	Position	: REAL	:= 0.0;	(* Actual Position *)
	Velocity	: REAL	:= 0.0;	(* Actual Velocity *)
	Torque		: REAL	:= 0.0;	(* Actual Torque *)
	Error		: UDINT	:= 0;	(* Error Code *)
	PowerActive	: BOOL  := FALSE;
	
END_STRUCT
END_TYPE

// ---- Data types/TF/Palletizer/TFMachinePalletizer_GatesAccess.TcDUT
TYPE TFMachinePalletizer_GatesAccess :
STRUCT
	GateAccessConsolle 	: TFGateAccess; //Consolle
	GateAccessPS306 	: TFGateAccessNoStop; //PS306 - Lato Sx Inizio
	GateAccessPS307 	: TFGateAccessNoStop; //PS307 - Lato Sx Centrale
	GateAccessPS308		: TFGateAccessNoStop; //PS308 - Lato Dx Centrale
	GateAccessPS309		: TFGateAccessNoStop; //PS309 - Lato DX In Fondo
END_STRUCT
END_TYPE

// ---- Data types/TF/Palletizer/TFMachinePalletizer_ManCmd.TcDUT
TYPE TFMachinePalletizer_ManCmd :
STRUCT
	CyclePallet : BOOL;
	CycleLayer : BOOL;
	Dest : INT;
	
	CicloRiposo	: BOOL;
	StepCiclo	: bool;
END_STRUCT
END_TYPE

// ---- Data types/TF/Palletizer/TFMachinePalletizer_ParametersFromHMI.TcDUT
TYPE TFMachinePalletizer_ParametersFromHMI :
STRUCT

	OffsetKPick					: REAL;	(* Offset di apertura pinza per prelievo pallet, falda  *)
	OffsetKPickPack				: REAL;	(* Offset di apertura pinza per prelievo pacco *)
	OffsetKPlacePack			: REAL;	(* Offset di apertura pinza per deposito pacco *)
	OffsetKPlace				: REAL;	(* Offset di apertura pinza per deposito pallet *)
	OffsetZPlacePallet			: REAL;	(* Offset quota Z per rilascio pallet *)
	OffsetZPlaceLayer			: REAL;	(* Offset quota Z per rilascio falda *)
	
	KPickTorquePallet			: REAL;	(* Coppia per prelievo Pallet *)
	
	OffsetZPlacePaccoVerticale		: REAL	:= 0; (* Offset quota Z per rilascio pacco in verticale *)
	OffsetZPlacePaccoOrrizzontale	: REAL 	:= 0;	(* Offset quota Z per rilascio pacco in Orrizzontale *)
	
	OffsetZUscitaTasteggioPickPallet : REAL := 10; (* Offset dell'asse Z durante un tasteggio in prelievo Pallet: l'asse Z si muove di questo offset dopo la ri-lettura dei tastatori *)

END_STRUCT
END_TYPE

// ---- Data types/TF/Palletizer/TFMachinePalletizer_WorkAreaOffset.TcDUT
(* Offset di posizionamento, rispetto alla posizione assoluta, delle postazioni nelle varie direzioni*)
TYPE TFMachinePalletizer_WorkAreaOffset :
STRUCT
	X : REAL := 0;	//Offset in direzione X
	Y : REAL := 0;	//Offset in direzione Y
	Z : REAL := 0;	//Offset in direzione Z
	RX : REAL := 0;	//Offset di rotazione lungo X
	RY : REAL := 0;	//Offset di rotazione lungo Y
	RZ : REAL := 0;	//Offset di rotazione lungo Z
END_STRUCT
END_TYPE

// ---- Data types/TF/Palletizer/TFMachinePalletizer_WorkAreaSort.TcDUT
TYPE TFMachinePalletizer_WorkAreaSort :
STRUCT
	Distance : LREAL;
	cwa : UINT;
END_STRUCT
END_TYPE

// ---- Data types/TF/Palletizer/TFMachinePalletizer_WorkAreaZone.TcDUT
TYPE TFMachinePalletizer_WorkAreaZone :
STRUCT
	Zone		: ARRAY[1..MAXZONE] OF TFMachinePalletizer_Zone; (* Definizione Zone *)
END_STRUCT
END_TYPE

// ---- Data types/TF/Palletizer/TFMachinePalletizer_WorkPickPointState_OLD.TcDUT
TYPE TFMachinePalletizer_WorkPickPointState_OLD :
STRUCT
	
	State			: INT	:= 0;	(* Stato PickPoint (0=Pacco Assente, 1=Pacco Presente *)
	Code			: INT	:= 0;	(* Codice Pacco *)
	NextCode		: INT	:= 0;   (* Codice Pacco Successivo *)
	TC				: INT   := 0;   (* Comando Ribaltino 0=Nop, 1=Ribaltino Verticale, 2=Ribaltino Orizzontale *)
	TS				: INT	:= 0;   (* Stato Ribaltino; 0=Nop,1=Ribaltino Verticale, 2=Ribaltino Orizzontale *)
	NextTC			: INT	:= 0;   (* Comando Successivo Ribaltino; 0=Nop, 1=Ribaltino Verticale, 2=Ribaltino Orizzontale*)
	ZTilter			: REAL  := 0.0; (* Quota asse Ribaltino, Scritta dall'Handling *)
	Encumbrance		: BOOL	:= FALSE; (* TRUE:= Le dimensioni del pacco sono tali da impegnare anche la PX di Uscita del Deviatore, FALSE:= Pacco cCmpletamente sul Ribaltino*)
	
	XDim			: REAL;		(* (mm) Dimensione X del Pacco *)
	YDim			: REAL;		(* (mm) Dimensione Y del Pacco *)
	ZDim			: REAL;		(* (mm) Dimensione Z del Pacco *)
	
END_STRUCT
END_TYPE

// ---- Data types/TF/Palletizer/TFMachinePalletizer_WorkPPOffset.TcDUT
TYPE TFMachinePalletizer_WorkPPOffset :
STRUCT
	Xv	:	REAL := 0.0; (* READ	- (mm) Offset del punto di prelievo in direzione X per ribaltino verticale *)
	Yv	:	REAL := 0.0; (* READ	- (mm) Offset del punto di prelievo in direzione Y per ribaltino verticale *)
	Zv	:	REAL := 0.0; (* READ	- (mm) Offset del punto di prelievo in direzione Z per ribaltino verticale *)
	Jv	:	REAL := 0.0; (* READ	- (mm) Offset di rotazione J  per ribaltino verticale *)
	
	Xh	:	REAL := 0.0; (* READ	- (mm) Offset del punto di prelievo in direzione X per ribaltino orrizontale *)
	Yh	:	REAL := 0.0; (* READ	- (mm) Offset del punto di prelievo in direzione Y per ribaltino orrizontale *)
	Zh	:	REAL := 0.0; (* READ	- (mm) Offset del punto di prelievo in direzione Z per ribaltino orrizontale *)
	Jh	:	REAL := 0.0; (* READ	- (mm) Offset di rotazione J per ribaltino orrizontale  *)
END_STRUCT
END_TYPE

// ---- Data types/TF/Palletizer/TFMachinePalletizer_Zone.TcDUT
TYPE TFMachinePalletizer_Zone :
STRUCT
	
	WorkArea	: ARRAY[1..MAXAREA] OF INT; 			(* Numero delle WorkArea *)
	Code		: ARRAY[1..MAXFORMINGCODE] OF INT;		(* Codici di Pallettizzazione (0..n=, -1 dato non valido) *)
	
END_STRUCT
END_TYPE

// ---- Data types/TF/Palletizer/TFModulePalletizerRobot_TCPPar.TcDUT
TYPE TFModulePalletizerRobot_TCPPar :
STRUCT
	
	X	: LREAL := 0;	(* READ	- X Axe Parameters (UI Position=mm, UI Velocity=mm/sec UI Acc/Dec=mm/sec2) *)
	Y	: LREAL := 0;	(* READ	- Y Axe Parameters (UI Position=mm, UI Velocity=mm/sec UI Acc/Dec=mm/sec2) *)
	Z	: LREAL := 0;	(* READ	- Z Axe Parameters (UI Position=mm, UI Velocity=mm/sec UI Acc/Dec=mm/sec2) *)
	
END_STRUCT
END_TYPE

// ---- Data types/TF/Palletizer/TFModulePalletizerRobot_Point.TcDUT
TYPE TFModulePalletizerRobot_Point :
STRUCT
	
	X				: REAL	:= 0.0;	(* X Position *)
	Y				: REAL	:= 0.0;	(* Y Position *)
	Z				: REAL	:= 0.0;	(* Z Position *)
	J				: REAL	:= 0.0;	(* J Position *)
	
END_STRUCT
END_TYPE

// ---- Data types/TF/Palletizer/TFModulePalletizerRobot_ManCmd.TcDUT
TYPE TFModulePalletizerRobot_ManCmd :
STRUCT
	
	X	: TFMachinePalletizer_AxeManCmd;	(* X Axe Manual Command *)
	Y	: TFMachinePalletizer_AxeManCmd;	(* Y Axe Manual Command *)
	Z	: TFMachinePalletizer_AxeManCmd;	(* Z Axe Manual Command *)
	J	: TFMachinePalletizer_AxeManCmd;	(* J Axe Manual Command *)
	K	: TFMachinePalletizer_AxeManCmd;	(* K Axe Manual Command *)
	
	GeneralHome : BOOL;
	
	SuctionOn 	: BOOL;
	SuctionOff 	: BOOL;
	SuctionUp 	: BOOL;
	SuctionDown : BOOL;

	Pinza : TFMachinePalletizer_PinzaVentoseManCmd;
	
	PosizionamentoPinza0 	: BOOL; //Posizionamento pinza 0°
	PosizionamentoPinza90 	: BOOL; //Posizionamento pinza 90°
	PosizionamentoPinza180 	: BOOL; //Posizionamento pinza 180°

END_STRUCT
END_TYPE

// ---- Data types/TF/Palletizer/TFMachinePalletizer_AxeParameters.TcDUT
TYPE TFMachinePalletizer_AxeParameters :
STRUCT
	
	HomeDefine		: REAL	:= 0.0;	(* READ	- Home Define (Posizione di Azzeramento Encoder) *)
	HomePosition	: REAL	:= 0.0;	(* READ	- Home Position (Posizione di Home) *)
	MaxVelocity		: REAL	:= 0.0;	(* READ	- Max Velocity (Velocità Massima) *)
	MaxAcceleration	: REAL	:= 0.0;	(* READ	- Max Acceleration (Accelerazione Massima) *)
	MaxDeceleration	: REAL	:= 0.0;	(* READ	- Max Deceleration (Decelerazione Massima) *)
	MinPosition		: REAL	:= 0.0;
	MaxPosition		: REAL	:= 0.0;
	MaxTorque		: REAL	:= 0.0;
	ManSlowVelocity	: REAL	:= 0.0; (* READ - Manual Slow Velocity (% of MaxVelocity) *)
	ManFastVelocity	: REAL	:= 0.0; (* READ - Manual Fast Velocity (% of MaxVelocity) *)
	
END_STRUCT
END_TYPE

// ---- Data types/TF/Palletizer/TFMachinePalletizer_AxeManCmd.TcDUT
TYPE TFMachinePalletizer_AxeManCmd :
STRUCT
	
	Home	: BOOL	:= FALSE;	(* READ	- Home (Ricerca Posizione di Home) *)
	JogPos	: BOOL	:= FALSE;	(* READ	- Jog + *)
	JogNeg	: BOOL	:= FALSE;	(* READ	- Jog - *)
	JogFast	: BOOL	:= FALSE;	(* READ	- Jog +/- in Fast Speed *)
	
END_STRUCT
END_TYPE

// ---- Data types/TF/Palletizer/TFMachinePalletizer_AxeState.TcDUT
TYPE TFMachinePalletizer_AxeState :
STRUCT
	
	Position	: REAL	:= 0.0;	(* Actual Position *)
	Velocity	: REAL	:= 0.0;	(* Actual Velocity *)
	Torque		: REAL	:= 0.0;	(* Actual Torque *)
	Error		: UDINT	:= 0;	(* Error Code *)
	
END_STRUCT
END_TYPE

// ---- Data types/TF/Palletizer/TFModulePalletizerRobot_AxisPar.TcDUT
TYPE TFModulePalletizerRobot_AxisPar :
STRUCT
	
	X	: TFMachinePalletizer_AxeParameters;	(* READ	- X Axe Parameters (UI Position=mm, UI Velocity=mm/sec UI Acc/Dec=mm/sec2) *)
	Y	: TFMachinePalletizer_AxeParameters;	(* READ	- Y Axe Parameters (UI Position=mm, UI Velocity=mm/sec UI Acc/Dec=mm/sec2) *)
	Z	: TFMachinePalletizer_AxeParameters;	(* READ	- Z Axe Parameters (UI Position=mm, UI Velocity=mm/sec UI Acc/Dec=mm/sec2) *)
	J	: TFMachinePalletizer_AxeParameters;	(* READ	- J Axe Parameters (UI Position=°,  UI Velocity=°/sec  UI Acc/Dec=°/sec2) *)
	K	: TFMachinePalletizer_AxeParameters;	(* READ	- K Axe Parameters (UI Position=mm, UI Velocity=mm/sec UI Acc/Dec=mm/sec2) *)
	
END_STRUCT
END_TYPE

// ---- Data types/TF/Palletizer/TFMachinePalletizer_Forming_OLD.TcDUT
TYPE TFMachinePalletizer_Forming_OLD :
STRUCT
	
	Enable		: INT							:= -1;	(* READ			- Formatura Abilitata 0=no, 1=si, -1 dato non valido *)
	Code		: ARRAY[1..MAXFORMINGCODE] OF INT;		(* READ			- Codici di Pallettizzazione (0..n=, -1 dato non valido) *)
	Pallet		: INT							:= -1;	(* READ			- Tipo di pallet assegnato (0 = tipo 0, 1 = tipo 1, 2 = tipo 2,  …. , 0 / -1 dato non valido *)
	Layer		: INT							:= -1;	(* READ			- Tipo di falda dopo il pallet (0 = assente, 1 = tipo 1, 2 = tipo 2,  …. , -1 dato non valido *)
	NLayer		: INT							:= -1;	(* READ			- Numero di falde da depositare ad inizio pallettizzazione *)
	Tape		: INT							:= -1;	(* READ			- Da Nastrare (0=no, 1=si, -1= non valido) *)
	LGVAttr		: INT								:= -1;  (* READ			- Attributi LGV (0=no, 1=si, -1= non valido) *)
	
	PX			: REAL							:= 0.0;	(* READ			- (mm) Pack X Dimension - Dimensione X (valore nominale) del pacco ribaltato in posizione verticale(al momento definiti come orizzontali) *)
	PY			: REAL							:= 0.0;	(* READ			- (mm) Pack Y Dimension - Dimensione Y (valore nominale) del pacco ribaltato in posizione verticale *)
	PZ			: REAL							:= 0.0;	(* READ			- (mm) Pack Z Dimension - Dimensione Z (valore nominale) del pacco ribaltato in posizione verticale *)
	PIZ			: REAL							:= 0.0;	(* READ			- (mm) Pack Z Pick  Offset - Offset Prelievo in Z *)
	PLZ			: REAL							:= 0.0; (* READ			- (mm) Pack Z Place Offset - Offset Deposito in Z *)
	AX			: REAL							:= 0.0; (* READ			- (mm) Approach X Distance - Distanza Accostamento X *)
	AY			: REAL							:= 0.0; (* READ			- (mm) Approach Y Distance - Distanza Accostamento X *)
	AZ			: REAL							:= 0.0; (* READ			- (mm) Approach Z Distance - Distanza Accostamento X *)
	KLT			: REAL							:= 0.0;	(* READ			- (%)  Valore di Coppia in presa Longitudinale *)
	KTT			: REAL							:= 0.0;	(* READ			- (%)  Valore di Coppia in Presa Trasversale *)
	KM			: INT							:= 0;	(* READ			- Modo Presa Pacco: 1=Position, 2=Position+Torque *)

	PickPosition: INT							:= 0; 	(* READ 		- 0 = misto, 1 = verticale, 2 = orizzontale*)
	PackXP		: ARRAY[1..MAXFORMINGPACK] OF TFMachinePalletizer_FormingPack; (* Tabella Pacchi X Positiva - Usata quando la X di Prelievo è Maggiore rispetto la quota di destinazione "Posizione Pallet" *)
	PackXN		: ARRAY[1..MAXFORMINGPACK] OF TFMachinePalletizer_FormingPack; (* Tabella Pacchi X Negativa - Usata quando la X di Prelievo è Minore rispetto la quota di destinazione "Posizione Pallet" *)
	
	GUID		: UINT;
	RecipeCode 	: UINT;              (* codice Ricetta *)
	
END_STRUCT
END_TYPE

// ---- Data types/TF/Palletizer/TFMachinePalletizer_FormingPack_OLD.TcDUT
TYPE TFMachinePalletizer_FormingPack_OLD :
STRUCT
	
	JP			: INT							:= -1;	(* READ	- Tipo di presa (1 = Longitudinale (x), 0 = Trasversale (Y se Verticale, Z se Orizzontale), -1 = dato non valido) *)
	Grip		: INT							:= -1;	(* READ	- Tipo di presa (0 = Verticale, 1 = Orizzontale, -1 = dato non valido) *)
	Trajectory	: INT							:= -1;	(* READ	- Tipo di percorso (0, 1, 2, 3, …) (-1 dato non valido) *)
	Layer		: INT							:= -1;	(* READ	- Tipo di falda dopo il pacco (0 = assente, 1 = tipo 1, 2 = tipo 2,  …. , -1 dato non valido *)
	
	X			: REAL							:= 0.0;	(* READ	- (mm) Destination - Coordinata X *)
	Y			: REAL							:= 0.0;	(* READ	- (mm) Destination - Coordinata Y *)
	Z			: REAL							:= 0.0;	(* READ	- (mm) Destination - Coordinata Z *)
	J			: REAL							:= 0.0;	(* READ	- (°)  Destination - Coordinata J *)
	
END_STRUCT
END_TYPE

(*
//Trajectory :	
 1= standard deposito in diagonale
 2= standard deposito in diagonale specchiato rispetto x
 3=	standard deposito in diagonale specchiato rispetto y
 4= standard deposito in diagonale specchiato rispetto x e y


Layer : quando devo mettere la falda






*)

// ---- Data types/TF/Palletizer/TFMachinePalletizer_IN.TcDUT
TYPE TFMachinePalletizer_IN :
STRUCT
	Mode : Mode;
	
	PowerOk : BOOL;
	
	SensorAir : BOOL;
	Sensor24Volt : BOOL;
	
	PX_WorkArea : ARRAY [1..MAXAREA] OF BOOL;
	
	HandlingRun : BOOL;
	
	Y_BeltSafety : BOOL;
	Z_BeltSafety : BOOL;
	PX_GripPresence : BOOL;
			
	WD_Trasporti : BOOL; //Watch DOG da Trasporti
	
END_STRUCT
END_TYPE

// ---- Data types/TF/Palletizer/TFMachinePalletizer_Layer_OLD.TcDUT
TYPE TFMachinePalletizer_Layer_OLD :
STRUCT
	X			: REAL	:= 0.0;	(* READ	- (mm) Dimensione X *)
	Y			: REAL	:= 0.0;	(* READ	- (mm) Dimensione Y *)
	Z			: REAL	:= 0.0;	(* READ	- (mm) Dimensione Z *)
END_STRUCT
END_TYPE

// ---- Data types/TF/Palletizer/TFMachinePalletizer_OUT.TcDUT
TYPE TFMachinePalletizer_OUT :
STRUCT
	Run : BOOL;
	Warning : BOOL;
	Error : BOOL;
	Horn : BOOL;
	StartHorn : BOOL;

	PowerActive : BOOL;
	
	HomeDone : BOOL;
	
	StopTilterReq : BOOL;
	PowerOffTilterReq : BOOL;
	PowerOnTilterReq : BOOL;
	ResetTilterReq : BOOL;
	StartTilter : BOOL;
	
	ClockSegnalazioni : bool;//Clock per segnalazioni varie
	
	PowerActiveSIMULAZIONE : BOOL;
	
	ClockSegnalazioniAlternato	: BOOL;//Clock Segnalazioni  Alternato
	ResetSirenaSegnalazioni : BOOL; //Segnale di stop suoneria sirena 
END_STRUCT
END_TYPE

// ---- Data types/TF/Palletizer/TFMachinePalletizer_Pallet_OLD.TcDUT
TYPE TFMachinePalletizer_Pallet_OLD :
STRUCT
	X			: REAL	:= 0.0;	(* READ	- (mm) Dimensione X *)
	Y			: REAL	:= 0.0;	(* READ	- (mm) Dimensione Y *)
	Z			: REAL	:= 0.0;	(* READ	- (mm) Dimensione Z *)
END_STRUCT
END_TYPE

// ---- Data types/TF/Palletizer/TFMachinePalletizer_VelocityOverride.TcDUT
TYPE TFMachinePalletizer_VelocityOverride :
STRUCT
	
	Auto		: REAL	:= 0.0;	(* READ	- (%) In Auto *)
	Jog			: REAL	:= 0.0;	(* READ	- (%) In Jog *)
	Pack		: REAL	:= 0.0;	(* READ	- (%) With Pack   (Durante il deposito di un pacco  / con Pacco a bordo) *)
	Pallet		: REAL	:= 0.0;	(* READ	- (%) With Pallet (Durante il deposito di un Pallet / con Pallet a bordo) *)
	Layer		: REAL	:= 0.0;	(* READ	- (%) With Layer  (Durante il deposito di un Layer  / con Falda a bordo) *)
	PickRip		: REAL	:= 0.0; (* READ - (%) Grip Free (Durante il prelievo di un Layer, una Falda o un Pacco) *)
	
END_STRUCT
END_TYPE

// ---- Data types/TF/Palletizer/TFMachinePalletizer_WorkArea_OLD.TcDUT
TYPE TFMachinePalletizer_WorkArea_OLD :
STRUCT

	Enable			: INT	:= -1;	(* READ			- Postazione Abilitata 0=no, 1=si, -1 dato non valido *)
	Typology		: INT	:= -1;	(* READ			- Tipologia 1=Catasta Vuoti, 2=Pallet Singolo, 3=Falda, -1 dato non valido *)
	Pallet			: INT	:= -1;	(* READ			- Tipo di pallet assegnato (0 = tipo 0, 1 = tipo 1, 2 = tipo 2,  …. , 0 / -1 dato non valido. Usato se Typology=1 *)
	Layer			: INT	:= -1;	(* READ			- Tipo di falda dopo il pallet (0 = assente, 1 = tipo 1, 2 = tipo 2,  …. , -1 dato non valido. Usato se Typology=3 *)
	Code			: INT	:= -1;	(* READ/WRITE	- Codice di Pallettizzazione (0..n=, -1 dato non valido). Viene estratto dalla Forming se Jolly=1, altrimenti lo si riceve! *)
	Jolly			: INT	:= -1;	(* READ/WRITE	- (Definizione del Codice di Pall... A carico del PLC) (0=no, 1=si, -1= non valido) *)
	Learn_Z			: REAL	:= 0.0;	(* READ			- (mm) Quota inizio Apprendimento "TouchProbe" Cataste e Falde) (Quota assoluta di impianto DA ORIGINE *)
	Learned_Z		: REAL	:= 0.0; (* WRITE		- Quota rilevata durante apprendimento *)
	DoLearn_Z			: INT	:= -1;	(* READ/WRITE 	- Stato apprendimento 0=Disabilitato, 1=Abilitato da Eseguire, 2=Eseguito, -1 dato non valido *)
	Slow			: INT	:= -1;	(* READ			- Primo Pacco in Lento (0=no, 1=si, -1= non valido) *)
	Taped			: INT	:= -1;	(* READ/WRITE	- Nastratura eseguita. Determina espulsione! (0=non eseguita, 1=eseguita, -1= non valido) *)
	RefuseLGV       : BOOL	:= FALSE;	(* READ		- Abilitazione chiamata LGV a termine pallettizzazione - TRUE= Non chiama LGV quando pallet pieno, FALSE= viene eseguita richiesta LGV *)
	Initialize		: BOOL	:= FALSE; 	(* READ		- Deposito pallet e falda se prevista e non continua la pallettizzazione, TRUE= deposita pallet e falda e non continua pallettizzazione, FALSE= Esegue tutto il ciclo regolarmente*)
	
	X				: REAL	:= 0.0;	(* READ			- (mm) Quota assoluta di impianto DA ORIGINE *)
	Y				: REAL	:= 0.0;	(* READ			- (mm) Quota assoluta di impianto DA ORIGINE *)
	Z				: REAL	:= 0.0;	(* READ			- (mm) Quota assoluta di impianto DA ORIGINE *)
	J				: REAL	:= 0.0;	(* READ			- (°) Quota assoluta di impianto DA ORIGINE *)
	H				: REAL	:= 0.0; (* READ/WRITE	- (mm) Altezza Reale. Viene calcolata dal PLC dopo ogni prelievo (Vuoti o Falde) o deposito Pallet e durante la pallettizzazione *)
	HPL				: REAL	:= 0.0; (* READ/WRITE   - (mm) Altezza del pallett utilizzato + altezza layers utilizzati *)
	
	JPick			: REAL	:= 0.0;	(* READ			- (°) Quota rotazione pinza per prelievo (usata se la workarea è un magazziono pallet/falde) *)
	KPick			: REAL	:= 0.0;	(* READ			- (mm) Quota apertura pinza per prelievo (usata se la workarea è un magazziono pallet/falde) *)
	JPlace			: REAL	:= 0.0;	(* READ			- (°) Quota rotazione pinza per deposito pallet/falde *)
	
	LGV_Req			: INT	:= 0;	(* READ/WRITE	- Richiesta LGV (0=Nop, 1=Richiesta LGV, 2= Consenso Ingresso, -1= non valido) *)
	LGV_GetIn_GetOut: INT	:= -1;	(* WRITE		- Tipo Richiesta LGV  (0=Nop, 1=Richiesta Prelievo, 2= Richiesta Deposito, -1= non valido) *)	
	LGV_LetIn		: INT	:= -1;	(* READ			- Stato LGV (0=Nop, 1=Richiesta Ingresso, 2=Fine Ingresso, -1= non valido) *)
	LGV_Footprint	: INT	:= -1;	(* READ			- Presenza Ingombro Veicolo (0=Nessun Ingombro, 1=In Ingombro, -1= non valido) *)
	LGV_ReqAbort	: BOOL	:= FALSE; (* READ		- Aborto chimata LGV *)
	
	ProgressiveNr	: UDINT;
	
END_STRUCT
END_TYPE

// ---- Data types/TF/Palletizer/TFMachinePalletizer_WorkFootprint.TcDUT
TYPE TFMachinePalletizer_WorkFootprint :
STRUCT
	X			: REAL	:= 0.0;	(* READ	- (mm) Quota assoluta di impianto DA ORIGINE *)
	Y			: REAL	:= 0.0;	(* READ	- (mm) Quota assoluta di impianto DA ORIGINE *)
	Z			: REAL	:= 0.0;	(* READ	- (mm) Quota assoluta di impianto DA ORIGINE *)
	XDim		: REAL	:= 0.0;	(* READ	- (mm) Dimensione X *)
	YDim		: REAL	:= 0.0;	(* READ	- (mm) Dimensione Y *)
	ZDim		: REAL	:= 0.0;	(* READ	- (mm) Dimensione Z *)	
END_STRUCT
END_TYPE

// ---- Data types/TF/Palletizer/TFMachinePalletizer_WorkPickPoint_OLD.TcDUT
TYPE TFMachinePalletizer_WorkPickPoint_OLD :
STRUCT
	
	Xv					: REAL	:= 0.0;		(* READ	- (mm) Quota assoluta di impianto DA ORIGINE - CON RIBALTINO IN VERTICALE *)
	Yv					: REAL	:= 0.0;		(* READ	- (mm) Quota assoluta di impianto DA ORIGINE - CON RIBALTINO IN VERTICALE *)
	Zv					: REAL	:= 0.0;		(* READ	- (mm) Quota assoluta di impianto DA ORIGINE - CON RIBALTINO IN VERTICALE *)
	Jv					: REAL	:= 0.0;		(* READ	- (mm) Quota assoluta di impianto DA ORIGINE - CON RIBALTINO IN VERTICALE *)
	ZvRaise				: REAL  := 0.0; 	(* READ	- (mm) Quota di salita per uscire dall'ingombro - CON RIBALTINO IN VERTICALE *)
	
	Xh					: REAL	:= 0.0;		(* READ	- (mm) Quota assoluta di impianto DA ORIGINE - CON RIBALTINO IN ORIZZONTALE *)
	Yh					: REAL	:= 0.0;		(* READ	- (mm) Quota assoluta di impianto DA ORIGINE - CON RIBALTINO IN ORIZZONTALE *)
	Zh					: REAL	:= 0.0;		(* READ	- (mm) Quota assoluta di impianto DA ORIGINE - CON RIBALTINO IN ORIZZONTALE *)
	Jh					: REAL	:= 0.0;		(* READ	- (mm) Quota assoluta di impianto DA ORIGINE - CON RIBALTINO IN ORIZZONTALE *)
	ZhRaise				: REAL  := 0.0; 	(* READ	- (mm) Quota di salita per uscire dall'ingombro - CON RIBALTINO IN ORIZZONTALE *)
	
END_STRUCT
END_TYPE

// ---- Data types/TF/Palletizer/TFMachinePalletizer_WorkSpace.TcDUT
TYPE TFMachinePalletizer_WorkSpace :
STRUCT
	X			: REAL	:= 0.0;	(* READ	- (mm) Quota assoluta di impianto DA ORIGINE *)
	Y			: REAL	:= 0.0;	(* READ	- (mm) Quota assoluta di impianto DA ORIGINE *)
	Z			: REAL	:= 0.0;	(* READ	- (mm) Quota assoluta di impianto DA ORIGINE *)
END_STRUCT
END_TYPE

// ---- Data types/TF/Palletizer/TFModulePalletizerRobot_Status.TcDUT
TYPE TFModulePalletizerRobot_Status :
STRUCT
	
	X	: TFMachinePalletizer_AxeState;	(* X Axe State (UI Position=mm, UI Velocity=mm/sec UI Acc/Dec=mm/sec2) *)
	Y	: TFMachinePalletizer_AxeState;	(* Y Axe State (UI Position=mm, UI Velocity=mm/sec UI Acc/Dec=mm/sec2) *)
	Z	: TFMachinePalletizer_AxeState;	(* Z Axe State (UI Position=mm, UI Velocity=mm/sec UI Acc/Dec=mm/sec2) *)
	J	: TFMachinePalletizer_AxeState;	(* J Axe State (UI Position=°,  UI Velocity=°/sec  UI Acc/Dec=°/sec2) *)
	K	: TFMachinePalletizer_AxeState;	(* K Axe State (UI Position=mm, UI Velocity=mm/sec UI Acc/Dec=mm/sec2) *)
	
	GroupSegmentVelocity : LREAL;
	GroupSegmentID : UDINT;
	
	MachineAuto : BOOL;
	MachineRun : BOOL;
	MachineError : UDINT;
	MachineErrorExtra : UDINT;
	
	RobotError : UDINT;
	RobotErrorExtra : UDINT;

	
END_STRUCT
END_TYPE

// ---- Data types/TF/Palletizer/TFModulePalletizerRobot_IN.TcDUT
TYPE TFModulePalletizerRobot_IN :
STRUCT
	
	PX_Touch 			: BOOL;
	PX_TouchEmergency 	: BOOL;
	PX_SuctionCupsUp	: BOOL;
	PX_StackLayer		: BOOL;
	PX_StackPallet		: BOOL;
	PX_GripPresence		: BOOL;
	
	Y_BeltSafety		: BOOL;
	Z_BeltSafety		: BOOL;

END_STRUCT
END_TYPE

// ---- Data types/TF/Palletizer/TFModulePalletizerRobot_OUT.TcDUT
TYPE TFModulePalletizerRobot_OUT :
STRUCT

	EV_Suction			: BOOL;
	EV_SuctionCupsUp	: BOOL;
	EV_SuctionCupsDown	: BOOL;
	
END_STRUCT
END_TYPE

// ---- Data types/TF/Rulliere/Macchina/TFMachineTransportIN.TcDUT
TYPE TFMachineTransportIN :
STRUCT
	Mode : Mode;
	PowerOk : BOOL;
	SensorAir : BOOL;
	Sensor24Volt : BOOL;
END_STRUCT
END_TYPE

// ---- Data types/TF/Rulliere/Macchina/TFMachineTransportManCmd.TcDUT
TYPE TFMachineTransportManCmd :
STRUCT
END_STRUCT
END_TYPE

// ---- Data types/TF/Rulliere/Macchina/TFMachineTransportOUT.TcDUT
TYPE TFMachineTransportOUT :
STRUCT
	Run : BOOL;
	Warning : BOOL;
	Error : BOOL;
	Horn : BOOL;
	StartHorn : BOOL;

	PowerActive : BOOL;
	
	HomeDone : BOOL;
	
	ClockSegnalazioni : BOOL;//Clock per segnalazioni varie
	
END_STRUCT
END_TYPE

// ---- Data types/TF/Rulliere/Moduli/Cinghia/TFCinghiaManCmd.TcDUT
TYPE TFCinghiaManCmd :
STRUCT
	Ax 					: TFAxManCmd;
	ResetModulo 		: BOOL;
	Ax2 				: TFAxManCmd;
	AbilitaCmdTandem	: BOOL;
END_STRUCT
END_TYPE

// ---- Data types/TF/Rulliere/Moduli/Cinghia/TFCinghia_IN.TcDUT
TYPE TFCinghia_IN :
STRUCT
	
	FTC_Presenza1 			: BOOL; // Fotocellula Presenza 1 "INGRESSO"
	FTC_Presenza1Enable 	: BOOL; // Fotocellula Presenza 1 Abilitata
	
	FTC_Presenza2		 	: BOOL; // Fotocellula Presenza 2 "MEDIANA"
	FTC_Presenza2Enable 	: BOOL; // Fotocellula Presenza 2 Abilitata 
	
	FTC_Presenza3		 	: BOOL; // Fotocellula Presenza 3 "USCITA"
	FTC_Presenza3Enable		: BOOL; // Fotocellula Presenza 3 Abilitata 
	
	StopEsterno 		: BOOL;//Comando di stop rotazione dall'esterno
	ConsensoDaValle 	: BOOL;//Consenso rotazione per invio materiale a valle
	StopDaMacchina 		: BOOL;//Stop COmando da macchina, per tutti quei comandi che rimangono sempre in esecuzione
	
END_STRUCT
END_TYPE

// ---- Data types/TF/Rulliere/Moduli/Cinghia/TFBancoScelta_IN.TcDUT
TYPE TFBancoScelta_IN :
STRUCT
	
	FTC_Presenza1 			: BOOL; // Fotocellula Presenza 1 "INGRESSO"
	FTC_Presenza1Enable 	: BOOL; // Fotocellula Presenza 1 Abilitata
	
	FTC_Presenza2		 	: BOOL; // Fotocellula Presenza 2 "MEDIANA"
	FTC_Presenza2Enable 	: BOOL; // Fotocellula Presenza 2 Abilitata 
	
	FTC_Presenza3		 	: BOOL; // Fotocellula Presenza 3 "USCITA"
	FTC_Presenza3Enable		: BOOL; // Fotocellula Presenza 3 Abilitata 
	
END_STRUCT
END_TYPE

// ---- Data types/TF/Rulliere/Moduli/Cinghia/TFCinghia_OUT.TcDUT
TYPE TFCinghia_OUT :
STRUCT
		FTC_Presenza1 : BOOL;//Segnale della FTC 1 in senso marcia
		FTC_Presenza2 : BOOL;//Segnale della FTC 2 in senso marcia
		FTC_Presenza3 : BOOL;//Segnale della FTC 3 in senso marcia	
		
		ConsensoAMonte 			: BOOL;//Consenso scarico materiale per modulo a monte
		VelocitaUscitaAValle 	: REAL;//Velocità di rotazione per modulo a valle
		StopEsterno 			: BOOL;//comando di stop esterno per altri moduli
		RichiestaAValle			: bool;//Richiesta di scarico al modulo a valle

END_STRUCT
END_TYPE

// ---- Data types/TF/Rulliere/Moduli/Cinghia/TFCinghiaParameters.TcDUT
TYPE TFCinghiaParameters :
STRUCT
	ExtraLoadSpace 		: REAL := 100; //Spazio Extra per fermata su sensore in fase di carico	
	ExtraUnloadSpace 	: REAL := 200; //Spazio Extra per scarico rulliera 
	ExtraSpinta      	: real := 50; //Spazion aggiungiuntivo per spinta pallet in accoppiamento
	//Con Carico a bordo
	VelocitaCarico			: REAL := 20; // [%] Percentuale Velocità Con carico a bordo
	AccCarico				: REAL := 20; // [%] Percentuale Accelerazione Con carico a bordo
	DecCarico				: REAL := 20; // [%] Percentuale Decelerazione Con carico a bordo
	//Senza Carico a bordo
	VelocitaVuoto			: REAL := 50; // [%] Percentuale Velocità Senza carico a bordo 
	AccVuoto				: REAL := 50; // [%] Percentuale Accelerazione Senza carico a bordo
	DecVuoto				: REAL := 50; // [%] Percentuale Decelerazione Senza carico a bordo
	//Manulai
	VelocitaJog				: REAL := 50; // [%] Percentuale Velocità Manuale
	AccJog					: REAL := 50; // [%] Percentuale Accelerazione Manuale
	DecJog					: REAL := 50; // [%] Percentuale Decelerazione Manuale

	CorrezioneVelocitaInverter2PerTandem 		: REAL := 5;
	CorrezioneVelocitaInverter2PerTandemMonte 	: REAL := 5;

END_STRUCT
END_TYPE

// ---- Data types/TF/Rulliere/Moduli/Cinghia/TFBancoScelta_OUT.TcDUT
TYPE TFBancoScelta_OUT :
STRUCT
		FTC_Presenza1 : BOOL;
		FTC_Presenza2 : BOOL;
		FTC_Presenza3 : BOOL;	
		
		
END_STRUCT
END_TYPE

// ---- Data types/TF/Rulliere/Moduli/Cinghia/TFMoveParAXCinghia.TcDUT
TYPE TFMoveParAXCinghia :
STRUCT
	AccCarico				: REAL := 20; // [mm/s2] Accelerazione FASE carico 
	DecCarico				: REAL := 20; // [mm/s2] Decelerazione FASE carico 
	VelocitaCarico			: REAL := 20; // [mm/s] Velocità FASE carico 
	
	AccScarico				: REAL := 20; // [mm/s2] Accelerazione FASE scarico
	DecScarico				: REAL := 20; // [mm/s2] Decelerazione FASE scarico
	VelocitaScarico			: REAL := 20; // [mm/s] Velocità FASE scarico
	
	VelocitaVuoto			: REAL := 20; // [mm/s] Velocità Senza carico a bordo 
	AccVuoto				: REAL := 20; // [mm/s2] Accelerazione Senza carico a bordo
	DecVuoto				: REAL := 20; // [mm/s2] Decelerazione Senza carico a bordo

	JerkConCarico			: REAL := 99999; //Jerk Con carico
	JerkVuoto				: REAL := 99999; //Jerk a Vuoto

END_STRUCT
END_TYPE

// ---- Data types/TF/Rulliere/Moduli/RullieraPallet/TFAxCentratoreManCmd.TcDUT
TYPE TFAxCentratoreManCmd :
STRUCT
	
	Home	: BOOL	:= FALSE;	(* Home (Ricerca Posizione di Home) *)
	JogPos	: BOOL	:= FALSE;	(* Jog + *)
	JogNeg	: BOOL	:= FALSE;	(* Jog - *)
	JogFast	: BOOL	:= FALSE;	(* Jog +/- in Fast Speed *)
	
	EseguiApertura 		: BOOL := FALSE; (* Porta il centratore tutto aperto *)
	EseguiCentratura 	: BOOL := FALSE; (* Esegue il ciclo di centratura *)
	
END_STRUCT
END_TYPE

// ---- Data types/TF/Rulliere/Moduli/RullieraPallet/TFAxTraslazioneRulliera.TcDUT
TYPE TFAxTraslazioneRulliera :
STRUCT
	
	Home	: BOOL	:= FALSE;	(* Home (Ricerca Posizione di Home) *)
	JogPos	: BOOL	:= FALSE;	(* Jog + *)
	JogNeg	: BOOL	:= FALSE;	(* Jog - *)
	JogFast	: BOOL	:= FALSE;	(* Jog +/- in Fast Speed *)
	
	MoveToCarico : BOOL := FALSE; (* Vai a posizione di CARICO*)
	MoveToScarico : BOOL := FALSE; (* Vai a posizione di CARICO*)
	MoveToPrelievo1 : BOOL := FALSE; (* Vai a posizione di CARICO*)
	MoveToPrelievo2 : BOOL := FALSE; (* Vai a posizione di CARICO*)
	
END_STRUCT
END_TYPE

// ---- Data types/TF/Rulliere/Moduli/RullieraPallet/TFCentratoreManCmd.TcDUT
TYPE TFCentratoreManCmd :
STRUCT
	Ax : TFAxCentratoreManCmd;
	ResetModulo : bool;	
END_STRUCT
END_TYPE

// ---- Data types/TF/Rulliere/Moduli/RullieraPallet/TFCentratoreParameters.TcDUT
TYPE TFCentratoreParameters :
STRUCT
	SogliaCentraturaEseguita	: REAL := 20; //Spazio Extra per fermata su sensore in fase di centratura	
	AbilitaCentratore			: bool := true; //Abilitazione centratore
	
	//Chiusura
	VelocitaChiusura		: REAL := 20; // [%] Percentuale Velocità chiusura(fino a sensori)
	VelocitaPareggiatura	: REAL := 20; // [%] Percentuale Velocità pareggiatura
	AccChiusura				: REAL := 20; // [%] Percentuale Accelerazione chiusura
	DecChiusura				: REAL := 20; // [%] Percentuale Decelerazione chiusra
	//Apertura
	VelocitaApertura		: REAL := 100; // [%] Percentuale Velocità apertura 
	AccApertura				: REAL := 100; // [%] Percentuale Accelerazione apertura
	DecApertura				: REAL := 100; // [%] Percentuale Decelerazione apertura
	
	//Manulai
	VelocitaJog				: REAL := 50; // [%] Percentuale Velocità Manuale
	AccJog					: REAL := 50; // [%] Percentuale Accelerazione Manuale
	DecJog					: REAL := 50; // [%] Percentuale Decelerazione Manuale

END_STRUCT
END_TYPE

// ---- Data types/TF/Rulliere/Moduli/RullieraPallet/TFCentratoreStatus.TcDUT
TYPE TFCentratoreStatus :
STRUCT

	Homed 		: BOOL; //Home modulo eseguito
	Error 		: UDINT; //Errore mofulo
	ErrorExtra 	: UDINT; //Errore extra modulo
	PowerActive : BOOL; //Modulo in marcia
	
	Ax1_State : TFMachinePalletizer_AxeState_weintek; //Stato asse 1
	
	Px_Home : BOOL; //Sensore reset
	Px_Aperto : BOOL; //Sensore extracorsa aperto
	Px_Chiuso : BOOL; //Sensore extracorsa chiuso

	Px_TouchDX : BOOL; //Sensore bandella DX
	Px_TouchSX : BOOL; //Sensore Bandella SX
	
	CentratoreAperto : BOOL;//Indica che il centratore è aperto in fuori ingombro
	
END_STRUCT
END_TYPE

// ---- Data types/TF/Rulliere/Moduli/RullieraPallet/TFCentratore_IN.TcDUT
TYPE TFCentratore_IN :
STRUCT
	
	TouchDX	: BOOL; //Sensore Bandella DX 1
	TouchSX		: BOOL; //Sensore Bandella SX 1
	
	PX_Aperto : BOOL; //Sensore MASSIMA APERTURA 1
	PX_Chiuso : BOOL; //Sensosre MASSIMA CHIUSURA 1
	PX_Home   : BOOL; //Sensore HOME 1
		
END_STRUCT
END_TYPE

// ---- Data types/TF/Rulliere/Moduli/RullieraPallet/TFCentratore_OUT.TcDUT
TYPE TFCentratore_OUT :
STRUCT
	PosizioneAperta : BOOL; //Posizione centratore Aperta e fuori ingombro
	PosizioneChiusa : BOOL; //Posizione centratore Chiusa e in ingombro
	PosizioneIndefinita : BOOL; //Posizione centratore Indefinita	
	
	FuoriIngombroXCarico : BOOL;//Posizione che consente alla rulliera di caricare senza che l'elemento in transito collida col centratore
	FuoriIngombroXScarico : BOOL;//Posizione che consente alla rulliera di scaricare l'elemento senza problemi
		
	TuochDX_Filtrato : BOOL;//Segnale stato bandella DX 
	TuochSX_Filtrato : BOOL;//Segnale stato bandella SX  

	PosizioneUltimaCentratura : REAL := 1900;//Posizione ultima centratura
		
END_STRUCT
END_TYPE

// ---- Data types/TF/Rulliere/Moduli/RullieraPallet/TFMoveParAXCentratore.TcDUT
TYPE TFMoveParAXCentratore :
STRUCT
	AccChiusura				: REAL := 20; // [mm/s2] Accelerazione Chiusura
	DecChiusura				: REAL := 20; // [mm/s2] Decelerazione Chiusura
	VelocitaChiusura		: REAL := 20; // [mm/s] Velocità Chiusura
	VelocitaApertura		: REAL := 20; // [mm/s] Velocità Apertura
	AccApertura				: REAL := 20; // [mm/s2] Accelerazione Apertura
	DecApertura				: REAL := 20; // [mm/s2] Decelerazione Apertura
	Jerk					: REAL := 999999;
	MinChiusura				: REAL := 400; 	// Quota minima di posizionamento	
	MaxApertura				: REAL := 1000; // Quota massima di posizionamento

END_STRUCT
END_TYPE

// ---- Data types/TF/Rulliere/Moduli/RullieraPallet/TFMoveParAXRulliera.TcDUT
TYPE TFMoveParAXRulliera :
STRUCT
	AccCarico				: REAL := 20; // [mm/s2] Accelerazione CON carico 
	DecCarico				: REAL := 20; // [mm/s2] Decelerazione CON carico 
	VelocitaCarico			: REAL := 20; // [mm/s] Velocità CON carico 
	
	AccScarico				: REAL := 20; // [mm/s2] Accelerazione SENZA scarico
	DecScarico				: REAL := 20; // [mm/s2] Decelerazione SENZA scarico
	VelocitaScarico			: REAL := 20; // [mm/s] Velocità SENZA scarico
	
	VelocitaVuoto			: REAL := 20; // [mm/s] Velocità Senza carico a bordo 
	AccVuoto				: REAL := 20; // [mm/s2] Accelerazione Senza carico a bordo
	DecVuoto				: REAL := 20; // [mm/s2] Decelerazione Senza carico a bordo
	JerkCarico				: REAL := 99999; //Jerk Con carico
	JerkVuoto				: REAL := 99999; //Jerk a Vuoto

	VelocitaPareggiatura	: REAL := 20; // [mm/s] Velocità Senza carico a bordo 


END_STRUCT
END_TYPE

// ---- Data types/TF/Rulliere/Moduli/RullieraPallet/TFMoveParAXTraslazioneRulliera.TcDUT
TYPE TFMoveParAXTraslazioneRulliera :
STRUCT
	AccCarico				: REAL := 20; // [mm/s2] Accelerazione Con carico a bordo
	DecCarico				: REAL := 20; // [mm/s2] Decelerazione Con carico a bordo
	VelocitaCarico			: REAL := 20; // [mm/s] Velocità Con carico a bordo
	VelocitaVuoto			: REAL := 20; // [mm/s] Velocità Senza carico a bordo 
	AccVuoto				: REAL := 20; // [mm/s2] Accelerazione Senza carico a bordo
	DecVuoto				: REAL := 20; // [mm/s2] Decelerazione Senza carico a bordo
END_STRUCT
END_TYPE

// ---- Data types/TF/Rulliere/Moduli/RullieraPallet/TFRullieraManCmd.TcDUT
TYPE TFRullieraManCmd :
STRUCT
	Ax 					: TFAxManCmd;
	ResetModulo 		: BOOL;
	Ax2 				: TFAxManCmd;
	AbilitaCmdTandemRulliere	: BOOL;
END_STRUCT
END_TYPE

// ---- Data types/TF/Rulliere/Moduli/RullieraPallet/TFRullieraMobileManCmd.TcDUT
TYPE TFRullieraMobileManCmd :
STRUCT
	AxR : TFAxManCmd;
	AxR2 : TFAxManCmd;
	AxT	: TFAxTraslazioneRulliera;
	ResetModulo : BOOL;
END_STRUCT
END_TYPE

// ---- Data types/TF/Rulliere/Moduli/RullieraPallet/TFRullieraMobileStatus.TcDUT
TYPE TFRullieraMobileStatus :
STRUCT
	Homed 		: BOOL; //Home modulo eseguito
	Error 		: UDINT; //Errore modulo
	ErrorExtra 	: UDINT; //Errore extra modulo
	PowerActive : BOOL; //Modulo in marcia
		
	Ax1_State : TFMachinePalletizer_AxeState_weintek; //Stato asse 1
	Ax2_State : TFMachinePalletizer_AxeState_weintek; //Stato Asse 2

	AxT_State : TFMachinePalletizer_AxeState_weintek; //Stato Asse Traslazione
	
	Element : TFMachineTransportElementWeintek;
	ElementPresente : BOOL;
	Element2 : TFMachineTransportElementWeintek;
	Element2Presente : BOOL;
	
	FTC_1 : BOOL; //Sensore 1
	FTC_2 : BOOL; //Sensore 2			
	FTC_3 : BOOL; //Sensore 3

	Px_Positivo : BOOL;//Sensore Extra corsa Positivo
	Px_Negativo : BOOL;//Sensore Extra corsa Positivo

	PosizioneRulliera : UINT; //Indica la posizione della rulliera

	StatoComando : UDINT;//Inidca lo stato in cui si trova il modulo

END_STRUCT
END_TYPE

// ---- Data types/TF/Rulliere/Moduli/RullieraPallet/TFRullieraParameters.TcDUT
TYPE TFRullieraParameters :
STRUCT
	ExtraLoadSpace 		: REAL := 100; //Spazio Extra per fermata su sensore in fase di carico	
	ExtraUnloadSpace 	: REAL := 200; //Spazio Extra per scarico rulliera 
	ExtraSpinta      	: real := 50; //Spazion aggiungiuntivo per spinta pallet in accoppiamento
	//Con Carico a bordo
	VelocitaCarico			: REAL := 20; // [%] Percentuale Velocità Con carico a bordo
	AccCarico				: REAL := 20; // [%] Percentuale Accelerazione Con carico a bordo
	DecCarico				: REAL := 20; // [%] Percentuale Decelerazione Con carico a bordo
	//Senza Carico a bordo
	VelocitaVuoto			: REAL := 50; // [%] Percentuale Velocità Senza carico a bordo 
	AccVuoto				: REAL := 50; // [%] Percentuale Accelerazione Senza carico a bordo
	DecVuoto				: REAL := 50; // [%] Percentuale Decelerazione Senza carico a bordo
	//Manulai
	VelocitaJog				: REAL := 50; // [%] Percentuale Velocità Manuale
	AccJog					: REAL := 50; // [%] Percentuale Accelerazione Manuale
	DecJog					: REAL := 50; // [%] Percentuale Decelerazione Manuale

	CorrezioneVelocitaInverter2PerTandem 		: REAL := 5;
	CorrezioneVelocitaInverter2PerTandemMonte 	: REAL := 5;

END_STRUCT
END_TYPE

// ---- Data types/TF/Rulliere/Moduli/RullieraPallet/TFRullieraStatus.TcDUT
TYPE TFRullieraStatus :
STRUCT

	Homed 		: BOOL; //Home modulo eseguito
	Error 		: UDINT; //Errore modulo
	ErrorExtra 	: UDINT; //Errore extra modulo
	PowerActive : BOOL; //Modulo in marcia
		
	Ax1_State : TFMachinePalletizer_AxeState_weintek; //Stato asse 1
	Ax2_State : TFMachinePalletizer_AxeState_weintek; //Stato Asse 2
	
	Element : TFMachineTransportElementWeintek;
	ElementPresente : BOOL;
	Element2 : TFMachineTransportElementWeintek;
	Element2Presente : BOOL;
	
	FTC_1 : BOOL; //Sensore 1
	FTC_2 : BOOL; //Sensore 2			
	FTC_3 : BOOL; //Sensore 3

	StatoComando : UDINT;//Inidca lo stato in cui si trova il modulo
	
END_STRUCT
END_TYPE

// ---- Data types/TF/Rulliere/Moduli/RullieraPallet/TFRulliera_IN.TcDUT
TYPE TFRulliera_IN :
STRUCT
	
	FTC_Presenza1 			: BOOL; // Fotocellula Presenza 1 "INGRESSO"
	FTC_Presenza1Enable 	: BOOL; // Fotocellula Presenza 1 Abilitata
	
	FTC_Presenza2		 	: BOOL; // Fotocellula Presenza 2 "MEDIANA"
	FTC_Presenza2Enable 	: BOOL; // Fotocellula Presenza 2 Abilitata 
	
	FTC_Presenza3		 	: BOOL; // Fotocellula Presenza 3 "USCITA"
	FTC_Presenza3Enable		: BOOL; // Fotocellula Presenza 3 Abilitata 
	
END_STRUCT
END_TYPE

// ---- Data types/TF/Rulliere/Moduli/RullieraPallet/TFRulliera_OUT.TcDUT
TYPE TFRulliera_OUT :
STRUCT
		FTC_Presenza1 : BOOL;
		FTC_Presenza2 : BOOL;
		FTC_Presenza3 : BOOL;	
		
		
END_STRUCT
END_TYPE

// ---- Data types/TF/Rulliere/Moduli/RullieraPallet/TFTraslazioneRullieraParameters.TcDUT
TYPE TFTraslazioneRullieraParameters :
STRUCT
	QuotaRullieraCarico 	: REAL := 100; //Posizione Rulliera di ingresso materiale	
	QuotaRullieraScarico 	: REAL := 2000; //Posizione Rulliera di uscita materiale
	QuotaRullieraPrelievo1 	: REAL := 100; //Posizione Rulliera di prelievo 1
	QuotaRullieraPrelievo2 	: REAL := 2000; //Posizione Rulliera di prelievo 2
	//Con Carico a bordo
	VelocitaCarico			: REAL := 20; // [%] Percentuale Velocità Con carico a bordo
	AccCarico				: REAL := 20; // [%] Percentuale Accelerazione Con carico a bordo
	DecCarico				: REAL := 20; // [%] Percentuale Decelerazione Con carico a bordo
	//Senza Carico a bordo
	VelocitaVuoto			: REAL := 50; // [%] Percentuale Velocità Senza carico a bordo 
	AccVuoto				: REAL := 50; // [%] Percentuale Accelerazione Senza carico a bordo
	DecVuoto				: REAL := 50; // [%] Percentuale Decelerazione Senza carico a bordo

	//Manulai
	VelocitaJog				: REAL := 50; // [%] Percentuale Velocità Manuale
	AccJog					: REAL := 50; // [%] Percentuale Accelerazione Manuale
	DecJog					: REAL := 50; // [%] Percentuale Decelerazione Manuale

END_STRUCT
END_TYPE

// ---- Data types/TF/Rulliere/Moduli/RullieraPallet/TFTraslazioneRulliera_IN.TcDUT
TYPE TFTraslazioneRulliera_IN :
STRUCT
	PX_Positive : BOOL; //Sensore Positivo
	PX_Negative : BOOL; //Sensore Negativo
	PX_Home   : BOOL; //Sensore HOME 
END_STRUCT
END_TYPE

// ---- Data types/TF/Rulliere/Moduli/TFAxManCmd.TcDUT
TYPE TFAxManCmd :
STRUCT
	
	Home	: BOOL	:= FALSE;	(* Home (Ricerca Posizione di Home) *)
	JogPos	: BOOL	:= FALSE;	(* Jog + *)
	JogNeg	: BOOL	:= FALSE;	(* Jog - *)
	JogFast	: BOOL	:= FALSE;	(* Jog +/- in Fast Speed *)
	
END_STRUCT
END_TYPE

// ---- Data types/TF/Rulliere/Moduli/TFAxParameters.TcDUT
TYPE TFAxParameters :
STRUCT
	HomeDefine		: REAL	:= 0.0;	(* Home Define (Posizione di Azzeramento Encoder) *)
	HomePosition	: REAL	:= 0.0;	(* Home Position (Posizione di Home) *)
	Vel				: REAL	:= 0.0;	(* Velocità di funzionamento*)
	Acc				: REAL	:= 100.0; (* Accelerazione di funzionamento *)
	Dec				: REAL	:= 100.0; (* Decelerazione di funzionamento *)
	Jerk			: REAL  := 100.0; (* Jerk di funzionamento *) 
	MaxTorque		: REAL	:= 100.0; (* Coppia massima utilizzata se si effettua il controllo di coppia*)
	JOGVel			: REAL	:= 100.0; (* Velocità JOG *)
	JOGAcc			: REAL	:= 100.0; (* Accelerazione JOG *)
	JOGDec 			: REAL	:= 100.0; (* Decelerazione JOG *)
	MaxDeceleration : REAL  := 100.0; (* Massima Decelerazione *)
	MinPosition		: REAL	:= 0.0;
	MaxPosition		: REAL	:= 0.0;
	MaxVel		    : REAL  := 0.0; (* Massima velocità per gestire i jog manuali *)
	MaxAcc		    : REAL  := 0.0; (* Massima velocità per gestire i jog manuali *)
	MaxDec		    : REAL  := 0.0; (* Massima velocità per gestire i jog manuali *)
	ManSlowVel		: REAL	:= 0.0; (* Manual Slow Velocity (% of MaxVelocity) *)
	ManFastVel		: REAL	:= 0.0; (* Manual Fast Velocity (% of MaxVelocity) *)
	Quota_Destinazione	: LREAL  := 0.0; (*Posizione target da raggiungere*)
	HomeVelocity		: REAL  := 1.0; (* Velocità per ricerca sesore di Home *)
END_STRUCT
END_TYPE

// ---- Data types/TF/Rulliere/Moduli/TFPortaStatus.TcDUT
TYPE TFPortaStatus :
STRUCT
	PortaAperta 	: BOOL;
	PortaChiusa 	: BOOL;
	AnomaliaPorta 	: BOOL;
END_STRUCT
END_TYPE

// ---- Data types/TF/Rulliere/Moduli/TFPortaManCmd.TcDUT
TYPE TFPortaManCmd :
STRUCT
	ApriPorta : BOOL;
	ChiudiPorta : bool;
END_STRUCT
END_TYPE

// ---- Data types/TF/Rulliere/Moduli/TFGestioneFTC_Misura_OUT.TcDUT
TYPE TFGestioneFTC_Misura_OUT :
STRUCT
	FTC_ZoccoloBassoFiltrata 	: BOOL;
	FTC_PallettoneFiltrata   	: BOOL;
	FTC_CavallinaBassaFiltrata 	: BOOL;
	FTC_CavallinaAltaFiltrata 	: BOOL;		

	LunghezzaMisurata 	: REAL;

	Supporto : TFMachinePalletizer_Pallet;
	
	MisuraInCorso : BOOL;
	MisuraDone : BOOL;
	
END_STRUCT
END_TYPE

// ---- Data types/TF/Rulliere/Moduli/TFBarcodeStatus.TcDUT
TYPE TFBarcodeStatus :
STRUCT

	Error 		: UDINT; //Errore modulo
	ErrorExtra 	: UDINT; //Errore extra modulo
		
	StatoLettore : StatusDataLogic;//Stato del lettore barcode

END_STRUCT
END_TYPE

// ---- Data types/TF/Rulliere/Moduli/TFTransportModules.TcDUT
TYPE TFTransportModules :
STRUCT

	BancoScelta 			: TFModuleSorterBancoScelta2Motori;
	ModuloCinghie 			: ARRAY[1..6] OF TFModuleCinghia;
	Bancalino 				: ARRAY[1..2] OF TFModuleBancalino;
	RullieraDopoBancalino 	: ARRAY[1..2] OF TFModuleRulliera;
	RullieraPareggiatore 	: ARRAY[1..2] OF TFModuleRulliera;
	RullieraPrelievo 		: ARRAY[1..2] OF TFModuleRulliera;
	
END_STRUCT
END_TYPE

// ---- Data types/TF/Rulliere/Moduli/TFTransportModuleStatus.TcDUT
TYPE TFTransportModuleStatus :
STRUCT
	Homed : BOOL; //Home modulo eseguito
	Error : UDINT;
	ErrorExtra : UDINT;
	PowerActive : BOOL; //Modulo in marcia
END_STRUCT
END_TYPE

// ---- Data types/TF/Rulliere/TFDimensionElement.TcDUT
TYPE TFDimensionElement :
STRUCT
	(* Dimensioni *)
	XDim		: REAL							:= 0.0;	(* (mm) Dimensione X *)
	YDim		: REAL							:= 0.0;	(* (mm) Dimensione Y *)
	ZDim		: REAL							:= 0.0;	(* (mm) Dimensione Z *)
END_STRUCT
END_TYPE

// ---- Data types/TF/Rulliere/TFMachinePalletizer_Pallet_Weintek.TcDUT
TYPE TFMachinePalletizer_Pallet_Weintek :
STRUCT
	Tipologia	: INT	:= -1;  (* Indica la tipologia dell'elemento *)
	Code		: INT;	(* Codici Della *)
	XDim		: REAL	:= 0.0;	(* (mm) Dimensione X *)
	YDim		: REAL	:= 0.0;	(* (mm) Dimensione Y *)
	ZDim		: REAL	:= 0.0;	(* (mm) Dimensione Z Base Cavallina o Base Cassa *)
	HMAX		: REAL  := 0.0;	(* (mm) Altezza Massima dell'elemento telaio cavallina o sponde cassa *)
	
	AltezzaDenteRitenuta	: REAL := 0.0; 	(* (mm) Altezza del dente di ritenuta (per cavalletti) *)
	Spessore_DenteRitenuta	: REAL := 0.0;	(* (mm) Spessore del dente di ritenuta (per cavalletti) *)
	OffsetY_DenteRitenuta 	: REAL := 0.0;	(* (mm) Posizione del dente di ritenuta rispetto la quota Y del cavalletto (per cavalletti) *)
	
	OFSDE_X90 				: REAL := 0.0;	(* (mm) OFFSET di deposito direzione X, utilizzato per PALLET o CASSE *)
	OFSDE_Y90 				: REAL := 0.0;	(* (mm) OFFSET di deposito direzione Y, utilizzato per PALLET o CASSE *)
	OFSDE_Z90 				: REAL := 0.0;	(* (mm) OFFSET di deposito direzione Z, utilizzato per PALLET o CASSE *)
	OFSDE_J90 				: REAL := 0.0;	(* (mm) OFFSET di deposito direzione J, utilizzato per PALLET o CASSE *)
	
	OFSDE_X0 				: REAL := 0.0;	(* (mm) OFFSET di deposito direzione X, utilizzato per CAVALLETTI *)
	OFSDE_Y0 				: REAL := 0.0;	(* (mm) OFFSET di deposito direzione Y, utilizzato per CAVALLETTI *)
	OFSDE_Z0 				: REAL := 0.0;	(* (mm) OFFSET di deposito direzione Z, utilizzato per CAVALLETTI *)
	OFSDE_J0 				: REAL := 0.0;	(* (mm) OFFSET di deposito direzione J, utilizzato per CAVALLETTI *)
	
	OFSDE_X180 				: REAL := 0.0;	(* (mm) OFFSET di deposito direzione X, utilizzato per CAVALLETTI *)
	OFSDE_Y180 				: REAL := 0.0;	(* (mm) OFFSET di deposito direzione Y, utilizzato per CAVALLETTI *)
	OFSDE_Z180 				: REAL := 0.0;	(* (mm) OFFSET di deposito direzione Z, utilizzato per CAVALLETTI *)
	OFSDE_J180 				: REAL := 0.0;	(* (mm) OFFSET di deposito direzione J, utilizzato per CAVALLETTI *)

	ConfigurazioneBC 	 : INT := -1;	(* (mm) Indica la modalità di funzionamento del barcode.. sono i suoi parametri *)
	QuotaRilevamentoBC_X : REAL := 0;	(* (mm) Indica la posizione del barcode lungo la sua lunghezza e rispetto il punto medio *)
	QuotaRilevamentoBC_Y : REAL := 0;	(* (mm) Indica la posizione del barcode lungo la sua larghezza e rispetto il punto medio	*)
	QuotaRilevamentoBC_Z : REAL := 0;	(* (mm) Indica la posizione del barcode lungo il suo spessore e rispetto il punto medio *)
	QuotaRilevamentoBC_J : REAL := 0;	(* (mm) Indica la posizione del barcode lungo il suo spessore e rispetto il punto medio *)

END_STRUCT
END_TYPE

// ---- Data types/TF/Rulliere/TFMachineTransportElement.TcDUT
TYPE TFMachineTransportElement :
STRUCT
	
	IDElement 		: UDINT := 0; //ID univoco generato dalla macchina  per il tracking degli alementi
	Barcode			: STRING := ''; //Barcode elemento
	DataElementOk 	: BOOL := FALSE;///Indica che i dati sono stati acquisiti e sono ok
	DataElement 	: TFMachinePalletizer_DataElement;
	DimElement 		: TFDimensionElement; //Dimensioni 
	Supporto		: TFMachinePalletizer_Pallet; (* Struttura del supporto presente sul punto di prelievo *)
	Zone			: e_ElementZone := e_ElementZone.NULL; //Zona di appartenenza dell'elemento
	ErrorAck		: BOOL := FALSE;//Se true, si attende un comando da parte dell'opperatore per far ripartire il ciclo
	CentraturaEsterna : e_StatoCentratura := CENTRATURA_DA_ESEGUIRE; //Stato della centratura estarna
	CentraturaInterna : e_StatoCentratura := CENTRATURA_DA_ESEGUIRE; //Stato della centratura interna
	Empty 				: BOOL := FALSE;	//Se TRUE significa che l'elemento è un vuoto
END_STRUCT
END_TYPE

// ---- Data types/TF/Rulliere/TFMachineTransportElementWeintek.TcDUT
TYPE TFMachineTransportElementWeintek :
STRUCT
	
	IDElement 		: UDINT := 0; //ID univoco generato dalla macchina  per il tracking degli alementi
	Barcode			: STRING := '';
	DataElementOk 	: BOOL := FALSE;///Indica che i dati sono stati acquisiti e sono ok
	DataElement 	: TFMachinePalletizer_DataElement;
	DimElement 		: TFDimensionElement; //Dimensioni 
	Supporto		: TFMachinePalletizer_Pallet_Weintek; (* Struttura del supporto presente sul punto di prelievo *)
	Zone			: INT := 0; //Zona di appartenenza dell'elemento
	ErrorAck		: BOOL := FALSE;//Se true, si attende un comando da parte dell'opperatore per far ripartire il ciclo
	CentraturaEsterna : INT; //Stato della centratura estarna
	CentraturaInterna : INT; //Stato della centratura interna
	Empty 			  : BOOL := FALSE;	//Se TRUE significa che l'elemento è un vuoto
END_STRUCT
END_TYPE

// ---- Data types/TF/Rulliere/TFMachineTransport_GatesAccess.TcDUT
TYPE TFMachineTransport_GatesAccess :
STRUCT
		
	GateAccessCarico 			: TFGateAccess;
	GateAccessCentratoreEsterno	: TFGateAccess;
	
END_STRUCT
END_TYPE

// ---- POUs/TFModules/DataBase/Record_From_DB.TcDUT
TYPE Record_From_DB :
STRUCT
	Udc 			: STRING(20);
	ArticleCode 	: STRING(20);
	Choice 			: STRING(5);
	Tone 				: STRING(5);
	Caliber 			: STRING(5);
	Length_mm 			: DINT;
	Width_mm 			: DINT;
	Thickness_mm 		: DINT;
	Quantity  			: LREAL;
	ArticleDescription 	: STRING(50);
END_STRUCT
END_TYPE

// ---- POUs/TFModules/DataBase/StoredProcedureState.TcDUT
TYPE StoredProcedureState :
STRUCT
	NumeroRecordLetti	: UDINT;//Numero di record letti
	ReadRun 		: BOOL;//Lettura in corso
	ReadDone 		: BOOL;//Lettura terminata con successo
	Error 			: BOOL;//Errore lettura
	ErrorID 		: UDINT;//ID Errore
	Sqlstate		: ST_DBSQLError;//State SQL
END_STRUCT
END_TYPE

// ---- POUs/TFModules/Misurazione Ingresso/TFGestioneFTC_Misura_IN.TcDUT
TYPE TFGestioneFTC_Misura_IN :
STRUCT
	FTC_ZoccoloBasso 	: BOOL;
	FTC_Pallettone   	: BOOL;
	FTC_CavallinaBassa 	: BOOL;
	FTC_CavallinaAlta 	: BOOL;
END_STRUCT
END_TYPE

// ---- Global Variables/BarCode/BarCODE.TcGVL
{attribute 'Tc2GvlVarNames'}
VAR_GLOBAL CONSTANT
	MAXNUMBARCODE		: INT := 4;		(* Identifica il numero dei BARCODE presenti nella WA (uno per ogni cassa nella WA) valorizza l'array dei BARCODE nella WASTATE *)
	DIMBARCODE			: INT := 13; 	(* Identifica la lunghezza del BARCODE *)

	(* Stati BARCODE *)
	LETTURA_DA_ESUGUIRE : INT := 0; 
	LETTURA_IN_CORSO 	: INT := 1;
	LETTURA_ESEGUITA 	: INT := 2;
	ERRORE				: INT := 3;
	
END_VAR

// ---- Global Variables/Comandi_1.TcGVL
{attribute 'Tc2GvlVarNames'}
VAR_GLOBAL CONSTANT
	
	CmdSbloccaBascolante 					: INT := 5000; (* Command: Do *)
	CmdBloccaBascolante 					: INT := 5100; (* Command: Do *)
	CmdSbloccaRotazione 					: INT := 5200; (* Command: Do *)
	CmdBloccaRotazione 						: INT := 5300; (* Command: Do *)
	CmdBloccaPinza							: INT := 5400; //blocco di tutta la pinza
	CmdSbloccaPinza							: INT := 5500; //sblocco di tutta la pinza

	
	StateSbloccaBascolante_RUN 			: INT := 5000;
	StateSbloccaBascolante_END 			: INT := 5099;
	StateBloccaBascolante_RUN 			: INT := 5100;
	StateBloccaBascolante_END 			: INT := 5199;
//                                        
	StateSbloccaRotazione_RUN 			: INT := 5200;
	StateSbloccaRotazione_END 			: INT := 5299;
	StateBloccaRotazione_RUN 			: INT := 5300;
	StateBloccaRotazione_END 			: INT := 5399;
                                          
	StateBloccaPinza_RUN 			: INT := 5400;
	StateBloccaPinza_END 			: INT := 5499;
	StateSbloccaPinza_RUN 			: INT := 5500;
	StateSbloccaPinza_END 			: INT := 5599;

	
END_VAR

// ---- Global Variables/Configurazione Impianto/Configurazione_Impianto.TcGVL
{attribute 'Tc2GvlVarNames'}
VAR_GLOBAL PERSISTENT
	(***********************************************************************************************************************************************************************************)
	(* Configurazioni comuni *)
	(***********************************************************************************************************************************************************************************)
	VERSO_PALLETTIZZATORE 				: e_Verso_Pallettizzatore 	:= PALLETTIZZATORE_SX; //Verso Pallettizzatore: stabilito guardando il pallettizzatore con la linea alle spalle
	TIPO_MAGAZZINO_FALDE  				: e_Tipo_Magazzino_Falde 	:= MAGAZZINO_FALDE_IN_WA; //Identifica il tipo di magazzino falde: MAGAZZINO_FALDE_CENTRO_FISSO = LA Y DI PRELIEVO RIMANE COSTANTE PER OGNI FORMATO,MAGAZZINO_FALDE_CENTRO_VARIABILE=LA Y DI PRELIEVO SI ADATTA AL FORMATO DELLA FALDA
	(***********************************************************************************************************************************************************************************)
	(* SOLO PER PALLETTIZZATORE LASTRE *)
	(***********************************************************************************************************************************************************************************)
	RIFERIMENTO_POSTAZIONE_WA			: e_RiferimentoPostazione 	:= CENTRALE; (*
												= 0		Identifica che la fotocellula di presenza della WorkArea è disposta sulla mediana della WorkArea stessa 	
												= 1 	Identifica che la fotocellula di presenza della WorkArea è disposta nell'angolo a SX della WorkArea stessa *)
	TIPOLOGIA_FUNZIONAMENTO_MACCHINA	: e_Tipo_Funzionamento := FUNZIONAMENTO_PICKING; (* Identifica la Tipolgia di funzionamento della Macchina *)											
	(***********************************************************************************************************************************************************************************)
	(* SOLO PER PALLETTIZZATORE PACCHI *)
	(***********************************************************************************************************************************************************************************)
	CATASTA_VUOTI_CON_RISCONTRI_FISSI 	: BOOL 						:= FALSE;	(*Se TRUE Identifica la presenza di riscontri fissi nella catasta dei vuoti (riscontri di centraggio) *)
	TIPO_RIBALTINO		  				: e_Tipo_Ribaltino 			:= RIBALTINO_DIRETTO;   (* Identifica il tipo di ribaltino (1= RIBALTINO DOPO SQUADRO,2= RIBALTINO DIRETTO) *)
	NPOSTAZIONE_DOPODELPUNTODIPREL		: UINT 						:= 5;		(* Numero Postazione DOPO del ribaltino ordine crescente di numero *)
	NPOSTAZIONE_PRIMADELPUNTODIPREL		: UINT 						:= 4;		(* Numero Postazione PRIMA del ribaltino, orfdine decrescente *)
	NumPostazionePALLET 				: INT; 									(* Indica il numero di postazione dove sono presenti I PALLET VUOTI *)
	(***********************************************************************************************************************************************************************************)
	(***********************************************************************************************************************************************************************************)
	NumPostazioneFALDE 					: UINT := 2; 							(* Indica il numero di postazione dove sono presenti LE FALDE *)
	NumPostazioneDiPareggiatura			: UINT := 3;							(* Indica il numero di postazione dove è presente la tavola di Pareggiatura *)

	ASSE_DISPOSIZIONE_POSTAZIONI		: e_Disposizione_Postazioni := LUNGO_X; (* Indica la disposizione delle postazioni rispeto gli assi della macchina, serve per capire la ciclica della macchina senza andare in collisione con le postazioni *)

	NUMERO_MACCHINA : UINT := 1; //Indica il numero della macchina in un impianto che usa la stessa HMI per discriminare eventuali pagine o funzioni in comune 

	ORDINE_DISPOSIZIONE_POSTAZIONI : e_OrdinamentoPostazione;// Indica come sono ordinate le postazioni rispetto l'origine della macchina: CRESCENTE o DECRESCENTE

	MAXAREAPRESENT : UINT := 4;//Piazzole di lavoro EFFETTIVAMENTE PRESENTI

	AngoloInclinazioneTavolaPareggiatura : REAL := 7; //Angolo in ° di inclinazione del della tavola di pareggiatura

	NumPostazioneBundle 	: UINT := 8;//Numero della postazione dedicata al bundle	
	AngoloInclinazioneBundle : REAL := 7; //Angolo in ° di inclinazione del del bundle

	NumPostazioneDeposito 	: UINT := 2;//Numero della postazione dedicata al deposito del materiale per pal picking
	NumPostazioneSuRulliera	: UINT := 1;//Numero della postazione dedicata al deposito del materiale per pal picking posizionata sulla rulliera
	

	
	HMaxScarto 			: REAL := 250;//Altezza massima ammissibile sul pancone degli scarti 
	CodeWasteSupport 	: INT := 4;	//Codice "Pallet dedicato al supporto degli scarti"
	
	TIPOLOGIA_RULLIERA_PRELIEVO : e_Tipologia_Rul_Prel;//Tipologia della ruliera di prelievo
	HMinFalde 			: REAL := 30;//Altezza minima sotto alla quale si manda in espulsione il pancone delle falde 
	CodeLayerSupport 	: INT := 15;	//Codice "Pallet dedicato al supporto delle falde"
	CodeWasteSlab		: INT := 3;//Codice lastra da scarare

	OFFSET_POSTAZIONE_LEGNO  : REAL := 680;//Offset filo fisso per legni rispetto al filo del bundle che è la quota di riferimento della WORKAREA lungo Y
	OFFSET_POSTAZIONE_TELAIO : REAL := 2630;//Offset filo fisso per TELAI rispetto al filo del bundle che è la quota di riferimento della WORKAREA lungo Y
	
	INGOMBRO_RISCONTRO_BUNDLE : REAL := 200;//Dimensione riscontro FISSO BUNDLE 
	INGOMBRO_RISCONTRO_FRAME : REAL := 100;//Dimensione riscontro FISSO BUNDLE 
END_VAR

VAR_GLOBAL CONSTANT

	(***********************************************************************************************************************************************************************************)
	(* SOLO PER PALLETTIZZATORE LASTRE *)
	(***********************************************************************************************************************************************************************************)
	//MAXPICKPOINTSTORE					: INT := 1;	(* Numero massimo di Punti di Prelievo di tipo Magazzino Falda *)
	//MAXPICKPOINTROLLER					: INT := 2;	(* Numero massimo di Punti di Prelievo di Tipo Rulliera *)
	(***********************************************************************************************************************************************************************************)
	(* SOLO PER PALLETTIZZATORE PACCHI *)
	(***********************************************************************************************************************************************************************************)
	ALTEZZA_CATASTA_VUOTI				: REAL := 1250;	(* Altezza Catasta Vuoti *)
	ALTEZZA_CATASTA_FALDE				: REAL := 900;	(* Altezza Catasta Falde *)
	
	DISTANZA_FTC_PINZA	: REAL := 650; (* Distanza tra le due fotocellule KEINCE sulla pinza *)

END_VAR

// ---- Global Variables/Errori/Errori_BarCODE.TcGVL
{attribute 'Tc2GvlVarNames'}
VAR_GLOBAL CONSTANT
	(* Errori BARCODE - CLASSE 6000 *)
	Err_TimeOUT_CmdBARCODE 	: INT := 6000;
	Err_TimeOUT_Lettura		: INT := 6001;

	ErrBARCODE_START : UINT := 13000;
	
	ErrBARCODE_1 : UINT:= ErrBARCODE_START +1;//Barcode non pronto, verficare connessione
	ErrBARCODE_2 : UINT:= ErrBARCODE_START +2;//Lettura Multipla, dato non valido
	ErrBARCODE_3 : UINT:= ErrBARCODE_START +3;//Timeout comando, anomalia nel sistema Barcode-FTC
	ErrBARCODE_4 : UINT:= ErrBARCODE_START +4;//Errore misurazione, lunghezza troppo corta
	ErrBARCODE_5 : UINT:= ErrBARCODE_START +5;//Barcode non letto
	ErrBARCODE_6 : UINT:= ErrBARCODE_START +6;//Scheduler ID mancante
	ErrBARCODE_7 : UINT:= ErrBARCODE_START +7;//Barcode già transitato/letto
	ErrBARCODE_8 : UINT:= ErrBARCODE_START +8;//Barcode non presente su DATABASE
	
END_VAR

// ---- Global Variables/Errori/Errori_CalcoloFormatura.TcGVL
{attribute 'Tc2GvlVarNames'}
VAR_GLOBAL
	
	ErrValori 				: UINT := 100;
	ErrHBaseInternaNulla 	: UINT := 101;
	ErrHBaseEsternaNulla 	: UINT := 102;
	ErrBaseInclinata 		: UINT := 103;
	ErrHTotaleNulla 		: UINT := 104;
	ErroreLBaseNulla 		: UINT := 105;
	ErrBase 				: UINT := 106;
	ErrLUtile 				: UINT := 107;
	ErrPendenzaBase 		: UINT := 108;
	ErrBaseAlfa 			: UINT := 109;
	ErrAltezzaAlfa 			: UINT := 110;
	ErrSpessoreZ 			: UINT := 111;
	ErrAngolo				: UINT := 112;
	ErrDimensioneCassa		: UINT := 113;
	ErrNumeroPezzi 			: UINT := 114;

	ErrNumeroMassimoFormatureAmmesse 	: UINT := 115;
	ErrRipetizioneCodici				: UINT := 116; //Errore in fase di attivazione: se sto attivando una formatura ma ce n'è un'altra attiva con i codici che si vogliono attivare 
	ErrNessunCodiciPresente				: UINT := 117; //Errore in fase di attivazione: se sto attivando una formatura che non ha nessn codice presente
	ErrDimensionesBundel				: UINT := 118;
	ErrDimensionCaballete				: UINT := 119 ;
	
	ErrDimensionCaballeteWa				: ARRAY [1..10] OF UINT  ;
	
	
END_VAR

// ---- Global Variables/Errori/Errori_WAManager.TcGVL
{attribute 'Tc2GvlVarNames'}
VAR_GLOBAL CONSTANT
	(* CLASSE 5000 *)
	ErrWAM_PickPoint_NoMagazzinoFalde 				: 	UINT := 5000; 	(* Il Pick Point che doveva essere un magazzino Falde, non è un magazzino falde *)
	ErrWAM_WorkArea_NoMagazzinoFalde 				: 	UINT := 5001; 	(* La WorkArea che doveva essere un magazzino Falde, non è un magazzino falde *)
	ErrWAM_TipologiaMagazzinoFaldaNONRiconosciuta 	: 	UINT := 5002;	(* La tipologia di magazzino falde impostata per l'impianto non è riconosciuta, 
																			definire se la tipologia di magazzino falde è di tipo PickPoint o WorkArea*)
	ErrWAM_TipologiaFaldaNONRiconosciuta			: 	UINT := 5003;	(* La tipologia di falda indicata non è presente nelle tipologia previste, 
																			definire una tipologia prevista (CARTONE,POLISTIROLO) *)
	ErrWAM_FaldeDepositateInEccesso					: 	UINT := 5004;	(* E' stato depositato un numero di falde superiore a quello previsto, RIMUOVERE manualmente la Falda Appena depositata e riprendere il ciclo Automatico*)																	
	ErrWAM_FaldaDepositataInWASbagliata				: 	UINT := 5005;	(* E' stato depositata una falda in una WA sbagliata, problema nella missione: non è stata calcolata correttamente o WAManager con Baco*)																	

	ErrWAM_TipologiaPalletNONRiconosciuta			: 	UINT := 5006;	(* E' stato depositata una falda in una WA sbagliata, problema nella missione: non è stata calcolata correttamente o WAManager con Baco*)																	

	ErrWAM_FTC_PostazioneNONDefinita				: 	UINT := 5007; 	(* La configurazione della FTC nella postazione non ha una definizione valida *)
	
	
	
	ErrWAM_FTCWA_ON_PrenzaLogicaOFF					: 	UINT := 5020; 	(* La FTC di presenza nella postazione è oscurata in modo anomalo senza che la macchina abbia la presenza LOGICA dell'elemento *)
	ErrWAM_FTCWA_OFF_PrenzaLogicaON				: 	UINT := 5021; 	(* La FTC di presenza nella postazione è spenta ma ho la presenza LOGICA dell'elemento *)

	//ErrWAM_FTCWA_ON_PrenzaLogicaOFF_bit				: 	ARRAY[1..MAXAREA] OF BOOL := FALSE; (* La FTC di presenza nella postazione è oscurata in modo anomalo senza che la macchina abbia la presenza LOGICA dell'elemento i-esimo *)

	ErrWAM_FTC_ON_PresenzaLastraPareggiatore		: UINT := 5022;		(* La FTC di presenza della lastra nella tavola di pareggiatura è oscurata in modo anomalo senza che la macchina abbia la presenza LOGICA dell'elemento *)
	ErrWAM_FTC_OFF_PresenzaLastraPareggiatore		: UINT := 5023; 	(* La FTC di presenza della lastra nella tavola di pareggiatura NON è oscurata e la macchina HA la presenza LOGICA dell'elemento,controllare FTC o eliminare LASTRA *)


	ErrWA_AnomaliaGestioneDepLastraDopoDepFalda 	: UINT := 5024; (* Dopo il deposito della falda, lo stato della pinza non mi permette di proseguire a causa di qualche condizione che non va, controllare lo stato della pinza e nel caso depositare la lastra a mano *)
	
	
	ErrWA_SupportoInPrelivoNonPrevisto				: UINT := 5025;  (* Il supporto sulla postazione in prelievo non è previsto *)
	ErrWA_SupportoInDepositoErrato					: UINT := 5026;  (* Il supporto sulla postazione di deposito non coincide col supporto richiesto dalla lista di lavoro *)
	ErrWA_NumPezzInPrelErrato						: UINT := 5027; (* Numero dei pezzi in prelievo < di 1, genero errore per evitare eccezioni *) 
	
END_VAR

// ---- Global Variables/Safety.TcGVL
{attribute 'Tc2GvlVarNames'}
VAR_GLOBAL

(* Variabili per uso Interno *)
	I_MarciaOK							AT %I* : BOOL; // Presenza marcia Ausiliari 
	I_EmergenzeOK						(*AT %I*) : BOOL; // Emergenze TUTTE ok

	I_BarrierePallettizzatoreOK			(*AT %I*) : BOOL; // Barriere TUTTE ok
	
	EnableGroupPortSafety 				AT %Q* : BOOL; 
	
	(* Stato FB Safety *)
	I_SafetyStateFunghiPal				AT %I* : USINT; //Stato FB Funghi Pallettizzatore
	I_SafetyStateBarrierDXPal			AT %I* : USINT; //Stato FB barriera Pallettizatore
	I_SafetyStateBarrierSXPal			AT %I* : USINT; //Stato FB barriera Pallettizatore
	I_SafetyStateBarrierCentroDXPal		AT %I* : USINT; //Stato FB barriera Pallettizatore
	I_SafetyStateBarrierCentroSXPal		AT %I* : USINT; //Stato FB barriera Pallettizatore
	I_SafetyStateBarrierKarv			AT %I* : USINT; //Stato FB barriera Pallettizatore
	I_SafetyStateEmergenze_Generali		AT %I* : USINT; //Stato FB Funghi Zona Bancalini

	//I_SafetyStateEmergenza_ConsollePS305	AT %I* : USINT; //Stato Fungo Consolle
	I_SafetyStateEmergenza_PS306_307			AT %I* : USINT; //Stato Fungo PS306
	I_SafetyStateEmergenza_PS308_309			AT %I* : USINT; //Stato Fungo PS307

	
	I_SafetyCOMERR						AT %I* : BOOL;  //Errore COM SAFETY 
	I_SafetyFBERR						AT %I* : BOOL;  //Errore FB SAFETY 
	I_SafetyOTHERERR					AT %I* : BOOL;  //Errore OTHER SAFETY 
	I_SafetyOUTERR						AT %I* : BOOL;  //Errore OUT SAFETY 

	I_SafetyCOMERR2						AT %I* : BOOL;  //Errore COM SAFETY 
	I_SafetyFBERR2						AT %I* : BOOL;  //Errore FB SAFETY 
	I_SafetyOTHERERR2					AT %I* : BOOL;  //Errore OTHER SAFETY 
	I_SafetyOUTERR2						AT %I* : BOOL;  //Errore OUT SAFETY 	

	O_AbilitazioneMarcia				AT %Q* : BOOL; //Abilitazione marcia a Centralina di sicurezza
	O_Reset_Plc_Sicurezza				AT %Q* : BOOL; //Comando di Reset PLC Sicurezza
	O_OverrideSoftwareBarriere_Pal		AT %Q* : BOOL := FALSE; //Override Software Barriere di sicurezza
	
	
	O_ResetACKAzionamenti AT%Q*:BOOL;
	
	I_FtcLGVPost_1 AT %I* : BOOL;//Ftc richiesta ingresso veicolo
	I_FtcLGVPost_2 AT %I* : BOOL;//Ftc richiesta ingresso veicolo
	I_FtcLGVPost_3 AT %I* : BOOL;//Ftc richiesta ingresso veicolo
	I_FtcLGVPost_4 AT %I* : BOOL;//Ftc richiesta ingresso veicolo
	I_FtcLGVPost_5 AT %I* : BOOL;//Ftc richiesta ingresso veicolo
	I_FtcLGVPost_6 AT %I* : BOOL;//Ftc richiesta ingresso veicolo
	I_FtcLGVPost_7 AT %I* : BOOL;//Ftc richiesta ingresso veicolo
	I_FtcLGVPost_8 AT %I* : BOOL;//Ftc richiesta ingresso veicolo
	
	O_RichiestaIngressoASafety AT %Q* : ARRAY[1..MAXAREA] OF BOOL;// Richiesta ingresso safety
	
	PortaleASx  : BOOL;//Il portale sta lavorando a SX e quindi l'operatore può entrare a DX
	PortaleADx  : BOOL;//Il portale sta lavorando a DX e quindi l'operatire può entrare a SX

END_VAR

VAR_GLOBAL CONSTANT
		
END_VAR

// ---- Global Variables/TFVariable/DATA_LOGGER.TcGVL
{attribute 'Tc2GvlVarNames'}
VAR_GLOBAL
	(* DataLogger *)
	DLogger : DataLogger();
	Channels : ARRAY [0..50] OF TFDataLogger.StatoCanaleRecord;
	DLOG_Cmd_ResetCounter 	: BOOL; //Resetta Tutti i contatori presenti 
	DLOG_Cmd_Alarm_reset 	: BOOL; //Resetta eventuali allarmi
	DLOG_Day_Reset : INT;
	DLOG_Week_Reset : INT := 7;
	DLOG_SaveDataOnReset : BOOL;
	Clogger : CounterLogger();
	Counters : ARRAY [0..50] OF TFDataLogger.StatoCanaleCounter;
	Reset_Operatore : BOOL;	// Comando da operatore di reset statistiche contattori
	Formign_ID_Active_Code : ARRAY [1..MAXFORMINGCODE] OF INT;	// Array per verifica formatura attiva su codice in verifica
	CLOG_Global_reset : BOOL;
END_VAR

// ---- Global Variables/TFVariable/Dati_Per_Linea.TcGVL
{attribute 'Tc2GvlVarNames'}
VAR_GLOBAL
	RichiestaDepositoALinea : BOOL;
	OkDepositoDaLinea		: BOOL;
	StateETHIPLinea			AT %I* : UINT;
	InputETHIPLinea 		AT %I* : ARRAY[1..50] OF WORD;
	OutputETHIPLinea 		AT %Q* : ARRAY[1..148] OF WORD;	
	DatiPerMP : TFMachinePalletizer_DataElementMP;

	DatiPalLinea : TFDatiDaLineaAPal;

END_VAR

// ---- Global Variables/TFVariable/FROM_HMI_PAL.TcGVL
{attribute 'Tc2GvlVarNames'}
VAR_GLOBAL PERSISTENT
(* Parametri assi del ciclo di riposo *)	
HMI_ParametriAsseX_CicloRiposo : Ax_Program_Parameters;	//Parametri dell'Asse X del ciclo di riposo
HMI_ParametriAsseY_CicloRiposo : Ax_Program_Parameters;	//Parametri dell'Asse Y del ciclo di riposo
HMI_ParametriAsseZ_CicloRiposo : Ax_Program_Parameters;	//Parametri dell'Asse Z del ciclo di riposo
HMI_ParametriAsseJ_CicloRiposo : Ax_Program_Parameters;	//Parametri dell'Asse J del ciclo di riposo
HMI_ParametriAsseK_CicloRiposo : Ax_Program_Parameters;	//Parametri dell'Asse K del ciclo di riposo
(* Parametri assi del ciclo falda *)
HMI_ParametriAsseX_CicloFalda : Ax_Program_Parameters;	//Parametri dell'Asse X del ciclo falda
HMI_ParametriAsseY_CicloFalda : Ax_Program_Parameters;	//Parametri dell'Asse Y del ciclo falda
HMI_ParametriAsseZ_CicloFalda : Ax_Program_Parameters;	//Parametri dell'Asse Z del ciclo falda
HMI_ParametriAsseJ_CicloFalda : Ax_Program_Parameters;	//Parametri dell'Asse J del ciclo falda
HMI_ParametriAsseK_CicloFalda : Ax_Program_Parameters;	//Parametri dell'Asse K del ciclo falda
(* Parametri assi del ciclo pallet *)
HMI_ParametriAsseX_CicloPallet : Ax_Program_Parameters;	//Parametri dell'Asse X del ciclo pallet
HMI_ParametriAsseY_CicloPallet : Ax_Program_Parameters;	//Parametri dell'Asse Y del ciclo pallet
HMI_ParametriAsseZ_CicloPallet : Ax_Program_Parameters;	//Parametri dell'Asse Z del ciclo pallet
HMI_ParametriAsseJ_CicloPallet : Ax_Program_Parameters;	//Parametri dell'Asse J del ciclo pallet
HMI_ParametriAsseK_CicloPallet : Ax_Program_Parameters;	//Parametri dell'Asse K del ciclo pallet
(* Parametri assi del ciclo pacco *)
HMI_ParametriAsseX_CicloPacco : Ax_Program_Parameters;	//Parametri dell'Asse X del ciclo pacco
HMI_ParametriAsseY_CicloPacco : Ax_Program_Parameters;	//Parametri dell'Asse Y del ciclo pacco
HMI_ParametriAsseZ_CicloPacco : Ax_Program_Parameters;	//Parametri dell'Asse Z del ciclo pacco
HMI_ParametriAsseJ_CicloPacco : Ax_Program_Parameters;	//Parametri dell'Asse J del ciclo pacco
HMI_ParametriAsseK_CicloPacco : Ax_Program_Parameters;	//Parametri dell'Asse K del ciclo pacco
(* Override delle varie modalità di funzionamento *)
HMI_AxisOverride : TFMachinePalletizer_VelocityOverride; //Override delle varie modalità di funzionamento
HMI_AbilitaControloPXGripPresence : BOOL := TRUE; // Variabile che abilita il controllo della fotocellula di presenza 
HMI_AbilitaControlloCoppia : BOOL := TRUE; // Variabile che abilita il controllo della fotocellula di presenza 
HMI_OffsetScattoAllarmeControlloCoppia : REAL := 10;
HMI_VelocitaDepositoPrimoPaccoInLenta : REAL := 50; // Velocità di deposito pacco, rispetto alla velocità standard, con la quale viene depositato il primo pacco dopo una modifica manuale del n° ei pacchi
HMI_VelocitaDiUscitaDaTastatoriAxZ	: REAL := 5; // Velocità dell'asse Z per uscire dai tastatori
HMI_AbilitaTasteggioDepositoPallet : Bool; // Abilitazione del tasteggio in fase di deposito pallet, in questo modo assegno la quota di altezza esatta alla piazzola
HMI_AbilitaForzaturaStatoDaRiposoAPrelievo : BOOL := FALSE; //Abilitazione della forzatura di passaggio di stato del WAM da Stato "Vai a riposo" a Stato "Pacco Init"
HMI_AbilitaDepositoPalletContinuo : BOOL := FALSE; //Abilitazione del deposito continuo dei pallet nel caso in cui il numero dei pacchi sia inferiore ad un certo valore
HMI_NumeroPacchiMassimoDepositoPalletContinuo : UINT := 7; // Valore al di sotto del quale si innesca il deposito dei pallet in continuo
HMI_OverideDinamico : Overide_Dinamico;	// Variabile per settare l'ovverride dinamico a soglie 
HMI_AbilitaOverrideDinamico : BOOL := FALSE; // Abilitazione della gestione automatica e dinamica dell'override
HMI_AbilitaAnticipoDinamicoMovimenti : BOOL := FALSE; // Abilitazione della gestione automatica delle quote per il comando dei movimenti
HMI_AbilitaComandiAnticipatiRibaltino : BOOL := FALSE; // Abilitazione della gestione avanzata del ribaltino
HMI_AbilitaDepositoPaccoOrrizzontaleConTasteggio : bool := false; // Abilitazione del deposito del pacco orrizzontale in modalità tasteggio
HMI_AbilitaInterpolazioneAssi : BOOL := FALSE; // Abilitazione dell'interpolazione degli assi
HMI_AbilitaGestioneAZone : BOOL := TRUE; //Abilitazione della gestione a zone delle WorkArea
HMI_VelocitaPercorso : REAL := 1000000000; // Velocità di percorrenza traiettoria con assi interpolati
HMI_TempoAccDec		 : REAL := 2; // Tempo di Accelerazione/Decelerazione dei movimenti nella traiettoria con assi interpolati
HMI_AbilitaOffsetUscitaTasteggioPrelPallet : BOOL := TRUE; // Abilitazione dell'offset in uscita dei tastatori in prelievo pallet con tasteggio
HMI_AbilitaCalcoloIngombroOttimizzato : BOOL := TRUE; // Abilitazione de calcolo degli ingombri in modo ottimizzato, valutando l'angolo di rotazione in tempo reale della pinza
HMI_AbilitaAccostamentoAsseZ : BOOL := TRUE; // Abilitazione dell'accostamento dell'asse Z.. Se TRUE : Ad una certa quota l'asse si muove in lenta 
HMI_AbilitaSimulazioneAVuoto : BOOL;//Abilitazione della simulazione senza pacchi-falde-pallet

HMI_AbilitaPosizionamentoDaQuoteApprese : BOOL; //Abilitazione del posizionamento utilizzando le quote ricavate in automatico dalla macchina

HMI_OvemParameters 				: Ovem_TargetParameters; //Parametri di funzionamento Vacuostato OVEM

HMI_AbilitaCilTastatoriPinza : BOOL;//Abilitazione dei tastatori della pinza
HMI_AbilitaSbloccoRotPinza : BOOL;//Abilitazione dello sblocco della rotazione della pinza
HMI_NumeroTentativiPresa :  UINT := 2;//numero di tentativi prima di dichiarare prelievo terminato
HMI_AbilitaTasteggioRotazionePinza : bool := true; //Abilitazione della ricerca automatica della posizione della rotazione mediante la distanza delle FTC di tasteggio
HMI_TempoPresaPiastrella : REAL := 2000;//Tempo per di attesa salita
HMI_VelocitaDiUscitaDaTastatoriAxY : real := 5;
HMI_OffsetUscitaTastatori : REAL := 2;
HMI_OffsetCompensazioneRotazionePinza : REAL := 5;

HMI_AbilitaSfogliaturaJ : BOOL := TRUE;
HMI_GradiSfogliaturaJ 	: REAL := 2;
 
HMI_TempoControlloPresaPiastrella 	: REAL := 500;//Tempo per il controllo di pistrella presa
HMI_TempoRilascioInDeposito 		: REAL := 500;//Tempo di attesa per distacco lastra in deposito
HMI_TempoAttesaPartenzaDopoPrelievo : REAL := 500;//Tempo di attesa per ripartenza dopo prelievo lastra
HMI_AbilitaAperturaAutomaticaPinza 	: BOOL;//Abilitazione apertura Automatica della pinza

HMI_ArrestoRullieraBancalino : BOOL;//Stop della rulliera su cui deposita la pinza
HMI_AbilitaPostazionePrelievo1 : BOOL;
HMI_AbilitaPostazionePrelievo2 : BOOL;

HMI_NumeroTentativiPolistiroloSuPallet : UINT := 2; //Indica il numero di tentativi di controllo sotto "HMI_AltezzaControlloPolistirolo" prima di espellere il pallet anche se risulta qualcosa in pinza che non sia una piastrella
HMI_AltezzaControlloPolistirolo : REAL := 0;//Indica la quota al di sotto della quale la macchina attiva il controllo di presenza se quota ripetuta

HMI_SpazioInterventoTastoriCartone : REAL := 30;

HMI_VelocitaDistaccoLastra_Z : REAL := 45;
HMI_VelocitaDistaccoLastra_Y : REAL := 10;

HMI_DisabilitaAsservimentoLGV : ARRAY[1..MAXAREA] OF BOOL;//Disabilitazione chiamata veicolo sulla postazione
HMI_AbilitaLettoreBC : bool; //Abilitazione lettore BC

HMI_TempoPresaFalda 						: REAL := 500;//Tempo di aggancio falda prima di risalire
HMI_TempoControlloPresaFalda 				: REAL := 500;//Tempo per il controllo di falda presa
HMI_TempoAttesaPartenzaDopoPrelievoFalda 	: REAL := 500;//Tempo di attesa per ripartenza dopo prelievo falda
HMI_TempoRilascioInDepositoFalda 			: REAL := 500;//Tempo di attesa per ripartenza dopo DEPOSITO falda
HMI_AbilitaDepositoFalda					: BOOL := TRUE; //ABilitazione deposito falda 

HMI_OffsetDepositoLastra	: ST_OffsetAllDirection;//Offset deposito lastra impostabile da HMI

HMI_OffsetGradiJPrelDaCanti				: REAL := 0;//Offset di inclinazione pinza x correzione posizione J in prelievo
HMI_AbilitaPosJPrelConFTC        : BOOL := TRUE;//Abilitazione del posizionamento J con le FTC poste sulla pinza

HMI_AbilitaBascolantePinza : bool;//Abilitazione del bascolante della pinza

END_VAR

VAR_GLOBAL
	HMI_AbilitazioneCicloAStep : BOOL := FALSE; // Variabile che abilita la modalità di funzionamento a step
	HMI_AbilitaErroriTastatori : BOOL := TRUE; // Variabile che abilita l'errore dovuto ai tastatori della pinza
	HMI_DisabilitaAnticipiGLOBALE : BOOL := TRUE; // Variabile per disabilitare tutti gli anticipi...si previene motion axis error 17035!!!!!!!!!
END_VAR

// ---- Global Variables/TFVariable/HMI_COMMAND_PAL.TcGVL
{attribute 'Tc2GvlVarNames'}
VAR_GLOBAL
	HMI_CommandSTEP : BOOL; // Comando dello step successivo con funzione ciclo in Step attivata
	
	HMI_AckBarcodeNonRiconosciuto : UINT;(*comando di gestione comportamento in caso di mancata lettura o lettura errata rispetto a quanto previsto
										 0= nessn comportamento, 1 =proseguo il ciclo e vado a depositare in postazione, 2 = vado a depositare in scarto*)

	HMI_Stop : BOOL;

	HMI_ForzaEspulsioneWA 	: ARRAY[1..MAXAREA] OF BOOL;//Variabile per forzare espulsione della postazione
	HMI_CodiceEspulsione	: ARRAY[1..MAXAREA] OF uint;//Varibile che identifica il codice di errrore da attribuire alla postazione, in questo modo si definisce la destinazione
	HMI_ManualClearWA 		: ARRAY[1..MAXAREA] OF BOOL;//Variabile per forzare pulizia postazione
	HMI_ManualRestoreWA 	: ARRAY[1..MAXAREA] OF BOOL;//Variabile per forzare ricreazione dati su postazione

END_VAR

// ---- Global Variables/TFVariable/HMI_Formatura.TcGVL
{attribute 'Tc2GvlVarNames'}
VAR_GLOBAL
	HMI_Forming_Calcola 					: BOOL; //START Esecuzione calcoli formatura
	HMI_Forming_Supporto 					: TFMachinePalletizer_Pallet; //Struttura pallet calcoli formatura
	HMI_Forming_LastraDaDepositare			: TFMachinePalletizer_PlaceElement; //Struttura dati dell'elemento da depositare 
	HMI_Forming_NumeroElementiDaDepositare 	: UINT; //Numero di elementi da depositare sul supporto

	HMI_Forming_FormaturaCalcolata			: TFMachinePalletizer_FormingForSlab; //Formatura calcolata dal FB
	HMI_Forming_ErroreCalcoli 				: UINT;//Errore calcoli formatura per sagnalazioni a operatore 
	
	HMI_Forming_ErroreCalcoliWa 			: ARRAY[1.. 12] OF UINT;//Errore calcoli formatura per sagnalazioni a operatore 
	
	HMI_Forming_IndiceFormaturaAttivata		: UINT; //Indica l'indice sul quale la formatura è stata attivata
	HMI_Forming_CodiciAbilitatiFormatura	: ARRAY[1..MAXFORMING] OF TFCodiciPerFormatura;

	HMI_Forming_GUID 						: UINT;
	HMI_Forming_Attivazione					: ARRAY[1..MAXFORMING] OF BOOL; //Attivazione formatura
	HMI_Forming_Disattivazione				: ARRAY[1..MAXFORMING] OF BOOL; //Disattiva formatura
	HMI_Forming_ErroreCalculos 				: ARRAY[1..MAXFORMING] OF BOOL; //Disattiva formatura
	
	HMI_Forming_FormaturaCreata 			:  BOOL; //TRUE se la formatura è stata creata correttamente
	HMI_Forming_FormaturaAttivata 			:  ARRAY[1..MAXFORMING] OF BOOL; //TRUE se la formatura è stata attivata correttamente
	HMI_Forming_FormaturaAttivataWa			:  ARRAY[1..MAXFORMING] OF BOOL;

	HMI_ErrAckCalcolaFormatura 				: BOOL; //Variabile che serve per dare ok acquisizione da operatore
	
	HMI_ConfermaAttivazioneFormatura		: ARRAY[1..MAXFORMING] OF BOOL;  //Bit per far uscire il popup di formatura attivata correttamente

	HMI_NumPostazioneSel					:INT ;
	HMI_ConfermaDati						:BOOL ;
	
	pippo : BOOL;

	
END_VAR

// ---- Global Variables/TFVariable/IO_TRASPORTI.TcGVL
{attribute 'Tc2GvlVarNames'}
VAR_GLOBAL CONSTANT
	MAXDIMARRAYPACCHI : UINT := 20; //Dimensione array dei pacchi sui trasporti
END_VAR

VAR_GLOBAL
	I_Trasporti_GEN_GLOBAL_ALARM_STOP 			(*AT %I**): BOOL; // Allarme Bloccante Trasporti
	I_Trasporti_PaccoSuRibaltino 				(*AT %I**) : DUT_Struttura_Dati_Pacco;  // Dati del Pacco SUl Ribaltino
	I_Trasporti_NumeroPacchiSuLinea 			(*AT %I**) : UINT; //Numero di pacchi presenti sulla linea
	I_Trasporti_NumeroUltimiTrasportiOccupati 	(*AT %I**) : UINT; //Numero degli ultimi trasporti occupati da un pacco
	                                            (*      *)
	I_Trasporti_GEN_ARRESTO_IN_FASE_ESEGUITO  	(*AT %I**): BOOL; //Stop in fase dei trasporti eseguito
	                                            (*      *)
	                                            (*      *)
	O_Trasporti_NumeroDiTrasportiDaValutare 	(*AT %Q**) : UINT; //Numero di trasporti da controllare
	O_Trasporti_GEN_RICH_ARRESTO_PALL 			(*AT %Q**) : BOOL; //Richiesta di stop in fase ai trasporti
	O_Centralina_Emergenze_Zona_Reggiatrice_OK	(*AT %Q**) : BOOL; //Sicurezze OK zona reggiatrice
	O_Centralina_Emergenze_Globali_OK			(*AT %Q**) : BOOL;	// Sicurezze globali OK - visualizzazione su pannello
	O_Centralina_Emergenze_PAL_OK 				(*AT %Q**) : BOOL;	// Sicurezze Pallettizzatore OK - gestione traini dentro a pal
	                                            (*      *)
	                                            (*      *)
	O_Trasporti_GEN_IN_RBT_WD 					(*AT %Q**) : BOOL;							// Segnale di wd
	O_Trasporti_GEN_IN_RBT_FI 					(*AT %Q**) : BOOL;							// Segnale di FI rbt
	O_Trasporti_GEN_IN_RBT_CMD_ORIZ 			(*AT %Q**) : BOOL;							// Segnale di ROTAZIONE ORIZZONTALE DA RBT
	O_Trasporti_GEN_IN_RBT_CMD_VERT 			(*AT %Q**) : BOOL;							// Segnale di ROTAZIONE VERTICALE DA RBT
	O_Trasporti_GEN_IN_RBT_AUTO 				(*AT %Q**) : BOOL;							// Stato auto robot
	O_Trasporti_EmergenzeOK						(*AT %Q**) : BOOL;							// Emergenze OK ai trasporti
	
	I_Trasporti_GEN_OUT_RBT_WD 						(*AT %I**) : BOOL;							// Segnale di wd
	I_Trasporti_GEN_OUT_PACCO_PRONTO_AL_PRELIEVO 	(*AT %I**) : BOOL;			// Bit segnalazione a RBT di prelievo pacco
	I_Trasporti_GEN_OUT_COMANDI_RBT_ABILITATI 		(*AT %I**) : BOOL;			// Bit segnalazione a RBT di Comandi disponibili
	I_Trasporti_GEN_OUT_RBT_LINEA_ARRESTO_IN_FASE 	(*AT %I**) : BOOL;		// Segnale Linea in arresto in fase
	I_Trasporti_GEN_OUT_AUTO_RBT 					(*AT %I**) : BOOL;					// Feedback sistema auto a robot
	I_Trasporti_GEN_QUOTA_RIBALTINO					(*AT %I**) : REAL;		// Quota ASSE Bandella attuale ribaltino
                                                    (*      *)
	I_Trasporti_GEN_OUT_ArrayPacchi 				(*AT %I**) :  DUT_ArrayPacchi; //Array Contenente i pacchi sui trasporti
	I_GEN_GLOBAL_ALARM_STOP							(*AT %I**) : Bool;//Indica che i trasporti sono in allarme
END_VAR

// ---- Global Variables/TFVariable/IO_Virtuali.TcGVL
{attribute 'Tc2GvlVarNames'}
VAR_GLOBAL
		
	(* LGV COMMUNICATION*)
	ILGV_LetIn								: BOOL;//	AT %I* : BOOL; Richiesta Ingresso DA LGV
	ILGV_Footprint							: BOOL;//	AT %I* : BOOL; LGV in Ingombro
	OLGV_Req								: BOOL;//	AT %I* : BOOL; Chiamata A LGV
	OLGV_LetIn								: BOOL;//	AT %I* : BOOL; Richiesta Ingresso DA LGV ricevuta e elaborata
	
	OLGV_ResetSW_RichiestaIngresso			(*AT %Q**) : BOOL;
	
	ILGV_LetIn_HW							(*AT %I**) : BOOL; //Richiesta Ingresso DA LGV segnale CABLATO
	ILGV_Footprint_HW						(*AT %I**) : BOOL; //LGV in INGOMBRO segnale CABLATO
	
	ILGV_LetIn_SW							: BOOL; //Richiesta Ingresso DA LGV segnale SOFTWARE
	ILGV_Footprint_SW						: BOOL; //LGV in INGOMBRO segnale SOFTWARE
	
	ISWITCH_HW_SW_LGV						: BOOL; //TRUE=segnale CABLATO,FALSE=segnale SOFTWARE
	
	O_PHConsensoIgressoNavetta				: ARRAY[1..MAXAREA] OF BOOL;
	I_PHPresenzaFalde				(*AT %I**) : BOOL;	//  = Fotocellula Presenza FALDE

	I_PHPresenzaMaterialePinza	: BOOL;
	I_EncoderX_Pronto	 		: BOOL;	// 16 = Encoder X Pronto
	I_24VAusiliariOK		 	: BOOL; 	// Presenza 24V ausiliari

END_VAR

// ---- Global Variables/TFVariable/LGV_Data.TcGVL
{attribute 'Tc2GvlVarNames'}
VAR_GLOBAL

	LGV_Stato_Pallettizzatore 	: LGV_Stato_Pallettizzatore;
	LGV_Stato_Postazione 		:  ARRAY [1..MAXAREA] OF LGV_Stato_Postazione;
	LGV_Stato_Formatura 		:  ARRAY [1..MAXFORMING] OF LGV_Stato_Formatura; 
	LGV_PostazioniPresenti 		: UINT;	//Indica il numero di postazioni presenti nel pallettizzatore (=MAXAREA)

	LGV_TipologiaSupervisore : INT := 0; //Indica la tipologia di protocollo utilizzata:0=Falomnet STANDARD,1=TECNOFERRARI
	(* Gestione Richieste Ingresso *)
	
	////////////////////////////////////////////////////////////////////////////////////////////////////////////////////////////////////////////////////////////////////////////////	
	(* Input *)
	I_LGV_CMD11_RichiestaIngresso		: BOOL; 	// Chiamata ingresso DA LGV,TRUE= La postazione è nello stato di chiamata navetta
	I_LGV_CMD11_InIngombro				: BOOL; 	// LGV in ingombro nella postazione
	(* Output *)
	O_LGV_CMD11_ChiamataDaMacchina	: BOOL; 	// Chiamata ingresso a LGV,TRUE=La una postazione è nello stato di chiamata navetta
	O_LGV_CMD11_OkIngressoMacchina 	: BOOL; 	// TRUE = OK Ingresso Nella Postazione 
		
	///////////////////////////////////////////////////////////////////////////////////////////////////////////////////////////////////////////////////////////////////////////////
	(* Input/Output *)
	I_LGV_Stato_Operazione : ARRAY [1..MAXAREA] OF INT; // Indica lo stato dell'operazione svolta dalla navetta: 0=Dato ricevuto e azzerato da PLC,1= Prelievo, 2= Deposito Concluso,
	O_LGV_Comando_Operazione  : ARRAY [1..MAXAREA] OF INT; // Indica il tipo di operazione che deve svolgere la navetta: 0=Nessuna operazione,1= Richieasta Prelievo, 2= Richiesta Deposito Vuoti,

	(* Input *)
	I_LGV_RichiestaIngresso		: ARRAY [1..MAXAREA] OF BOOL; 	// Chiamata ingresso DA LGV,TRUE= La postazione è nello stato di chiamata navetta
	I_LGV_InIngombro			: ARRAY [1..MAXAREA] OF BOOL; 	// LGV in ingombro nella postazione
    
	(* Output *)
	O_LGV_ChiamataDaPostazione		: ARRAY [1..MAXAREA] OF BOOL; 	// Chiamata ingresso a LGV,TRUE=La una postazione è nello stato di chiamata navetta
	O_LGV_OkIngressoInPostazione 	: ARRAY [1..MAXAREA] OF BOOL; 	// TRUE = OK Ingresso Nella Postazione 
	
	(* Configurazione segnali *)
	I_LGV_SegnaliCablati   : BOOL;		// LGV Seleziona la Tipologia di gestione segnali: TRUE=Segnali Cablati,FALSE=Segnali Software

	(* Segnali cablati *)
	I_LGV_RichiestaIngresso_HW	AT %I* : ARRAY [1..MAXAREA] OF BOOL; 	// Chiamata ingresso a LGV,TRUE=La postazione è nello stato di chiamata navetta
	I_LGV_InIngombro_HW			AT %I* : ARRAY [1..MAXAREA] OF BOOL;	// LGV in ingombro
	O_LGV_OKIngresso_HW			AT %I* : ARRAY [1..MAXAREA] OF BOOL; 	// TRUE = OK Ingresso Nella Postazione 
	///////////////////////////////////////////////////////////////////////////////////////////////////////////////////////////////////////////////////////////////////////////////

	O_LGV_ProductDataRequest : ARRAY [1..MAXAREA] OF TFMachinePalletizer_DataElement;//Dati per richiesta a supervisore materiale

	MachinePalletizerLGV : ARRAY [1..MAXAREA] OF GateAccessLGV; 	//FB di gestione richiesta ingresso veicolo

END_VAR

// ---- Global Variables/TFVariable/Picking.TcGVL
{attribute 'Tc2GvlVarNames'}
VAR_GLOBAL CONSTANT

	MAXPRODLIST			: UINT := 3; //Numero LISTE DI PRODUZIONE DA ESEGUIRE
	MAXARTICLEPICKING 	: UINT := 4; //Numero di "Prodotti" necessari per comporre l'ordine di picking.. corrisponde al numero di postazioni disponibili in macchina
	MAXELEMENTLIST 		: UINT := 100;//Numero massimo di elementi presenti nella lista di produzione -> N° falde+ N° lastre	
END_VAR

VAR_GLOBAL
	Cmd_CalcolaLista 	: ARRAY [1..3] OF BOOL;//Comando che crea la lista di produzione
	Cmd_AttivaLista 	: ARRAY [1..3] OF BOOL;//Comando attivazione nuova lista
	Cmd_AzzeraLista 	: ARRAY [1..3] OF BOOL; //Comando Reset Lista Attiva

	ListaInEsecuzione 		: ARRAY [1..3] OF BOOL; //Indica che una lista è già in esecuzione
	NumeroListaInEsecuzione : UINT;
	IdxMaxNumEl 			: UINT;
	ElementiDaDepositare 	: ARRAY [1..3] OF UINT;
	ElementiElaborati 		: ARRAY [1..3] OF UINT;
	HMI_NumeroLastreDepOrdineAttuale 		: ARRAY [1..3] OF UINT; //Numero lastre depositate ordine attuale
	HMI_NumeroLastreRimanentiOrdineAttuale 	: ARRAY [1..MAXAREA] OF UINT;//numero lastre rimanenti postazione di prelievo
	ListaEmpty 								: TFMachinePalletizer_ListaProduzione_WAM;
	SlabNumber								: INT;
END_VAR

VAR_GLOBAL PERSISTENT
	HMI_PareggiaturaLastraAbilitata : BOOL; //Abilitazione Pareggiatore lastre
	PickingListFROMSupervisorArray 	: ARRAY [1..MAXPRODLIST] OF TFMachinePalletizer_ListaProduzione;//Lista di produzione dal supervisore
	
	PickingListFROMSupervisor 		: TFMachinePalletizer_ListaProduzione;//Lista di produzione dal supervisore
	
	//ok sotto
	RequestPickingListFromHMI 			: ARRAY [1..3] OF ST_DataManualPicking;
	ActualPickingListFromHMI  			: ARRAY [1..3] OF ST_DataManualPicking;
	RequestPickingListFromHMIWorkArea  	: ARRAY [1..MAXAREA] OF ST_DataManualPicking;
		
	HMI_WorkAreaDataPicking 		: ARRAY [1..MAXAREA] OF ST_WorkAreaDataPicking;//Dati da HMI per definire il picking
	HMI_WorkLadoTrabajo_Cavallete	: INT ;// 0-trabaja aambos lados 1-Lado 0 Grados 2-Lado 180 Grados
	HMi_DimensionesPiezasWorkAreaDeposito	: ARRAY  [1..MAXELEMENTLIST] OF ES_dimensionPiezaLadoA_ladoB; 
	
	HMI_ErroreCalcoloLista : UINT := 0;//Errori utilizzati per il calcolo della lista
	
	//PickingListTOSupervisor 		: ARRAY [1..MAXPRODLIST] OF TFMachinePalletizer_ListaProduzione;//Lista di produzione a supervisore
	FormaturaBundleRT : ARRAY [1..3] OF TFMachinePalletizer_FormingForSlab; //Formatura real time di appoggio per calcoli di prel-dep in supporti non orizzontali
	FormaturaAFRAMERT : ARRAY [1..3] OF TFMachinePalletizer_FormingForSlab; //Formatura real time di appoggio per calcoli di prel-dep in supporti non orizzontali
	FormaturaWa		  : ARRAY [1..MAXAREA] OF TFMachinePalletizer_FormingForSlab;
	
	
	HMI_NumeroPezziPresentiPostazione 	: ARRAY [1..MAXAREA] OF UINT;
	HMI_NumeroPezziPresentiCavallete 	: ARRAY [1..MAXAREA] OF Es_PiezasCaballete;

	HMI_WorkAreaDataPicking_1_8 	: BOOL; //Ordine postazioni 1..8 in lavoro
	HMI_WorkAreaDataPicking_1_4 	: BOOL; //Ordine postazioni 1..4 in lavoro
	HMI_WorkAreaDataPicking_5_8 	: BOOL; //Ordine postazioni 1..4 in lavoro	
	
	Numero_Piezas_estacionPikin					: UINT;
	Numero_piezas_CaballeteEstacionPiking 		: Es_PiezasCaballete;
END_VAR

// ---- Global Variables/TFVariable/Pinza.TcGVL
{attribute 'Tc2GvlVarNames'}
VAR_GLOBAL

	(* VARIABILI OVEM DX*)	
	Ovem1 								: TF_VacumOVEM;
	ComunicazioneOvem1 					: Ovem_Comunication;
	I_LivelloDepressioneOVEM_BL_1 		AT %I* : WORD; //Proces Data BYTE LOW  Ovem
	I_LivelloDepressioneOVEM_BH_1 		AT %I* : WORD; //Proces Data BYTE HIGHT Ovem
	I_PortQualifierOVEM_1 				AT %I* : WORD; //Port Qualifier Ovem
	O_ControlWordOVEM_1 				AT %Q* : WORD; //Control Word Ovem A
	(* VARIABILI OVEM SX*)
	Ovem2 								: TF_VacumOVEM;
	ComunicazioneOvem2 					: Ovem_Comunication;
	I_LivelloDepressioneOVEM_BL_2 		AT %I* : WORD; //Proces Data BYTE LOW Ovem
	I_LivelloDepressioneOVEM_BH_2 		AT %I* : WORD; //Proces Data BYTE HIGHT Ovem
	I_PortQualifierOVEM_2 				AT %I* : WORD; //Port Qualifier Ovem
	O_ControlWordOVEM_2 				AT %Q* : WORD; //Control Word Ovem A
	
	CommandOVEM_1			: Ovem_Command;//Comandi Ovem 1
	CommandOVEM_2			: Ovem_Command;//Comandi Ovem 2
	
	(* VARIABILI OVEM DX2*)	
	Ovem12 								: TF_VacumOVEM;
	ComunicazioneOvem12 				: Ovem_Comunication;
	I_LivelloDepressioneOVEM_BL_12 		AT %I* : WORD; //Proces Data BYTE LOW  Ovem
	I_LivelloDepressioneOVEM_BH_12 		AT %I* : WORD; //Proces Data BYTE HIGHT Ovem
	I_PortQualifierOVEM_12 				AT %I* : WORD; //Port Qualifier Ovem
	O_ControlWordOVEM_12 				AT %Q* : WORD; //Control Word Ovem A
	(* VARIABILI OVEM SX2*)
	Ovem22 								: TF_VacumOVEM;
	ComunicazioneOvem22 				: Ovem_Comunication;
	I_LivelloDepressioneOVEM_BL_22 		AT %I* : WORD; //Proces Data BYTE LOW Ovem
	I_LivelloDepressioneOVEM_BH_22 		AT %I* : WORD; //Proces Data BYTE HIGHT Ovem
	I_PortQualifierOVEM_22 				AT %I* : WORD; //Port Qualifier Ovem
	O_ControlWordOVEM_22 				AT %Q* : WORD; //Control Word Ovem A
	
	CommandOVEM_12			: Ovem_Command;//Comandi Ovem 1
	CommandOVEM_22			: Ovem_Command;//Comandi Ovem 2

	CilindroAperturaPinza 	: DC_Cylinder;
	CilindroSbloccoPinza 	: SC_Cylinder;
	CilindroTasteggio 		: SC_Cylinder;
	AspirazioneFaldaDX 		: SC_Cylinder;
	AspirazioneFaldaSX 		: SC_Cylinder;
	CilindroSbloccoBascolante :  SC_Cylinder;

	PinzaVentoseManCmd : TFMachinePalletizer_PinzaVentoseManCmd;

	LetturaFTCPinza0_1 	 : REAL;
	LetturaFTCPinza180_1 : REAL;
	LetturaFTCPinza0_2 	 : REAL;
	LetturaFTCPinza180_2 : REAL;
	
	AlPosDestinoBandelCavaleta: REAL;
	
END_VAR

VAR_GLOBAL PERSISTENT

END_VAR

// ---- Global Variables/TFVariable/QE_BORDO.TcGVL
{attribute 'Tc2GvlVarNames'}
VAR_GLOBAL		

I_SicurezzaCinghia_Y	(*AT %I*) : BOOL;	// = Sicurezza Cinghia Y
I_SicurezzaCinghia_Z	(*AT %I*) : BOOL;	// = Sicurezza Cinghia Z

(* Ingressi su azionamenti *)
(* X-Y*)
I_ExtraCorsaNegativo_X 	(*AT %I*) : BOOL;  // 0 = Extra CorSa Negativo Asse X
I_ExtraCorsaPositivo_X 	(*AT %I*) : BOOL;  // 1 = Extra CorSa Negativo Asse X
I_ResetAsse_X 			(*AT %I*) : BOOL;  // 2 = Reset Asse X

I_ExtraCorsaNegativo_Y 	(*AT %I*) : BOOL;  // 4 = Extra CorSa Negativo Asse Y
I_ExtraCorsaPositivo_Y 	(*AT %I*) : BOOL;  // 5 = Extra CorSa Negativo Asse Y
I_ResetAsse_Y			(*AT %I*) : BOOL;  // 6 = Reset Asse Y

(* Z-K *)
I_ZKDriveDigitalInput							AT %I* : UINT;

I_ExtraCorsaNegativo_Z  (*AT %I*) : BOOL;  // 0 = Extra CorSa Negativo Asse Z
I_ExtraCorsaPositivo_Z  (*AT %I*) : BOOL;  // 1 = Extra CorSa Negativo Asse Z
I_ResetAsse_Z		    (*AT %I*) : BOOL;  // 2 = Reset Asse Z

I_ExtraCorsaNegativo_J  (*AT %I*) : BOOL;  // 0 = Extra CorSa Negativo Asse Z
I_ExtraCorsaPositivo_J  (*AT %I*) : BOOL;  // 1 = Extra CorSa Negativo Asse Z
I_ResetAsse_J		    (*AT %I*) : BOOL;  // 2 = Reset Asse Z

(* Singoli assi *)
I_XDriveDigitalInput	AT %I* : UDINT;
I_YDriveDigitalInput	AT %I* : UDINT;
I_ZDriveDigitalInput	AT %I* : UDINT;
I_JDriveDigitalInput	AT %I* : UDINT;

I_XDriveError			AT %I* : DWORD;
I_YDriveError			AT %I* : DWORD;
I_ZDriveError			AT %I* : DWORD;
I_JDriveError			AT %I* : DWORD;

O_XDriveDigitalOutput	AT %Q* : UINT;
O_YDriveDigitalOutput	AT %Q* : UINT;
O_ZDriveDigitalOutput	AT %Q* : UINT;
O_JDriveDigitalOutput	AT %Q* : UINT;

I_FermoSicurezzaRilasciato 	: BOOL;
O_SbloccoFermoSicurezza 	: BOOL; 

I_RotazioneColonnaBloccata 	: BOOL;
I_TastatoreBascolante		: BOOL;

////////// Ciabatte Bordo Pinza /////////////

(* J16 *)
O_AperturaPinza : BOOL; // X1.0 pin 4
O_ChiusuraPinza : BOOL; // X1.0 pin 2
O_SbloccoPinza 	: BOOL; // X1.1 pin 4

I_PinzaApertaDX	: BOOL; // 
I_PinzaChiusaDX	: BOOL; // 
I_PinzaApertaSX	: BOOL; // 
I_PinzaChiusaSX	: BOOL; // 
I_BascolantePinzaBloccato 	: BOOL; //K516-X1.4 pin 4
I_TasteggioCinghiaAsseZ 	: BOOL; //K516-X1.7 PIN 2

O_AspirazioneCartoneESTSX : BOOL; // X1.5 pin 4 - Aspirazione Cartone Esterno Lato SX
O_AspirazioneCartoneINTSX : BOOL; // X1.6 pin 4 - Aspirazione Cartone Interno Lato SX
O_AspirazioneCartoneESTDX : BOOL; // X1.7 pin 4 - Aspirazione Cartone Esterno Lato DX

I_TastoreCartone1 : BOOL; // X1.0 pin 4 - Presenza Falda Lato DX
I_TastoreCartone2 : BOOL; // X1.0 pin 2 - Presenza Falda Lato SX

I_TastatorePinza_1	(*AT %I*) : BOOL;	// X1.1 pin 4 - Tastatore Pinza 1
I_TastatorePinza_2	(*AT %I*) : BOOL;	// X1.1 pin 2 - Tastatore Pinza 2
I_TastatorePinza_3	(*AT %I*) : BOOL;	// X1.2 pin 4 - Tastatore Pinza 3
I_TastatorePinza_4	(*AT %I*) : BOOL;	// X1.2 pin 2 - Tastatore Pinza 4
I_TastatorePinza_5	(*AT %I*) : BOOL;	// X1.2 pin 4 - Tastatore Pinza 3
I_TastatorePinza_6	(*AT %I*) : BOOL;	// X1.2 pin 2 - Tastatore Pinza 4

I_TastatoreEmergenzaPinza_1	(*AT %I*) : BOOL;	// X1.3 pin 4 - Tastatore Emergenza Pinza 1
I_TastatoreEmergenzaPinza_2	(*AT %I*) : BOOL;	// X1.3 pin 2 - Tastatore Emergenza Pinza 2
I_TastatoreEmergenzaPinza_3	(*AT %I*) : BOOL;	// X1.4 pin 4 - Tastatore Emergenza Pinza 3
I_TastatoreEmergenzaPinza_4 (*AT %I*) : BOOL;	// X1.4 pin 2 - Tastatore Emergenza Pinza 4
I_TastatoreEmergenzaPinza_5	(*AT %I*) : BOOL;	// X1.4 pin 4 - Tastatore Emergenza Pinza 3
I_TastatoreEmergenzaPinza_6 (*AT %I*) : BOOL;	// X1.4 pin 2 - Tastatore Emergenza Pinza 4

I_PHPresenzaFaldaDX : BOOL; //J16 Porta 5 pin 2
I_PHPresenzaFaldaSX : BOOL; //J16 Porta 5 pin 4

I_ExtraCorsaPinzaSganciata : BOOL; // X1.6 pin 4 - Controllo della rotazione lungo z, extracora con pinza sganciata

//O_AspirazioneCartoneINTDX 	: BOOL; // X1.7 pin 4 - Aspirazione Cartone Interno Lato DX 
//O_AttivaTastatoriPinza		: BOOL; // X1.7 pin 2 - Aspirazione Cartone Interno Lato DX 

I_Keyence0_Byte0 	AT %I* : BYTE;
I_Keyence0_Byte1 	AT %I* : BYTE;
I_Keyence180_Byte0 	AT %I* : BYTE;
I_Keyence180_Byte1 	AT %I* : BYTE;

I_Keyence0_Byte0_2 	AT %I* : BYTE;
I_Keyence0_Byte1_2 	AT %I* : BYTE;
I_Keyence180_Byte0_2 	AT %I* : BYTE;
I_Keyence180_Byte1_2 	AT %I* : BYTE;


I_CiabattaPinzaK515AMSADDR 		AT %I* : AMSADDR;
I_TimeStampCiabattaPinzaK515 	AT %I* : ULINT;
I_CiabattaPinzaK516AMSADDR 		AT %I* : AMSADDR;
I_TimeStampCiabattaPinzaK516 	AT %I* : ULINT;
I_CiabattaPinzaK517AMSADDR 		AT %I* : AMSADDR;
I_TimeStampCiabattaPinzaK517 	AT %I* : ULINT;

I_K515_XO3 AT %I* : ARRAY[0..3] OF BYTE;
I_K515_XO4 AT %I* : ARRAY[0..3] OF BYTE;

I_K516_XO3 AT %I* : ARRAY[0..3] OF BYTE;
I_K516_XO4 AT %I* : ARRAY[0..3] OF BYTE;

//Q_K515 AT %Q* : ARRAY[0..31] OF BYTE;
//I_K516 AT %I* : ARRAY[0..31] OF BYTE;
//Q_K516 AT %Q* : ARRAY[0..31] OF BYTE;
I_K517 AT %I* : ARRAY[0..31] OF BYTE;
Q_K517 AT %Q* : ARRAY[0..31] OF BYTE;

I_PortQualCiabattaK515_X01 AT %I* : WORD;
I_PortQualCiabattaK515_X02 AT %I* : WORD;
I_PortQualCiabattaK515_X03 AT %I* : WORD;
I_PortQualCiabattaK515_X04 AT %I* : WORD;
I_PortQualCiabattaK515_X05 AT %I* : WORD;
I_PortQualCiabattaK515_X06 AT %I* : WORD;
I_PortQualCiabattaK515_X07 AT %I* : WORD;
I_PortQualCiabattaK515_X08 AT %I* : WORD;

I_PortQualCiabattaK516_X01 AT %I* : WORD;
I_PortQualCiabattaK516_X02 AT %I* : WORD;
I_PortQualCiabattaK516_X03 AT %I* : WORD;
I_PortQualCiabattaK516_X04 AT %I* : WORD;
I_PortQualCiabattaK516_X05 AT %I* : WORD;
I_PortQualCiabattaK516_X06 AT %I* : WORD;
I_PortQualCiabattaK516_X07 AT %I* : WORD;
I_PortQualCiabattaK516_X08 AT %I* : WORD;

I_PortQualCiabattaK517_X01 AT %I* : WORD;
I_PortQualCiabattaK517_X02 AT %I* : WORD;
I_PortQualCiabattaK517_X03 AT %I* : WORD;
I_PortQualCiabattaK517_X04 AT %I* : WORD;
I_PortQualCiabattaK517_X05 AT %I* : WORD;
I_PortQualCiabattaK517_X06 AT %I* : WORD;
I_PortQualCiabattaK517_X07 AT %I* : WORD;
I_PortQualCiabattaK517_X08 AT %I* : WORD;


END_VAR

// ---- Global Variables/TFVariable/QE_TERRA.TcGVL
{attribute 'Tc2GvlVarNames'}
VAR_GLOBAL
	
	//******************** SCHEDA IN AP200.2		
	I_AP200_2 			AT %I*: ARRAY[1..16] OF BOOL;

	I_AutoPal			: BOOL;	// 1 = Selettore manuale automatico Pal
	I_StartCicloPal		: BOOL;	// 2 = Star Ciclo Pallettizzatore
	I_StopCicloPal		: BOOL;	// 3 = Stop Ciclo Pallettizzatore
	//I_FREE 			: bool; // 4 = FREE
	//I_FREE 			: bool; // 5 = FREE
	I_AriaOK			: BOOL; // 6 = Aria ok 
	I_24VOK_AUXQE		: BOOL; // 7 = Presenza 24V AUSILIARI Quadro
	I_24VOK_SAFETY		: BOOL; // 8 = Presenza 24V SAFETY
	I_24VOK_MONITOR		: BOOL; // 9 = Presenza 24V MONITOR
	I_24VOK_PS305		: BOOL; // 10 = Presenza 24V PS305
	I_24VOK_PS306		: BOOL;	// 11 = Presenza 24V PS306
	I_24VOK_PS307		: BOOL;	// 12 = Presenza 24V PS307
	I_24VOK_JB310		: BOOL; // 13 = Presenza 24V JB311
	I_24VOK_JB311 		: BOOL; // 14 = Presenza 24V JB311
	I_24VOK_JB312 		: BOOL; // 15 = Presenza 24V JB312
	I_24VOK_JB313 		: BOOL; // 16 = Presenza 24V JB313

	//******************** SCHEDA IN SAFETY AP200.3		
	I_AP200_3 			AT %I*: ARRAY[1..4] OF BOOL;
	//I_EmergenzaGenerale_CH1 	: BOOL; // 1=
	//I_EmergenzaGenerale_CH2 	: BOOL; // 2=	
	//I_BarrieraDX_CH1			: BOOL; // 3=	
	//I_BarrieraDX_CH2			: BOOL; // 4=	

	//******************** SCHEDA IN SAFETY AP200.4		
	I_AP200_4 			AT %I*: ARRAY[1..4] OF BOOL;
	//I_EmergenzaPS306PS307_CH1 	: BOOL; // 1=
	//I_EmergenzaPS306PS307_CH2 	: BOOL; // 2=	
	//I_BarrieraPS308PS309_CH1		: BOOL; // 3=	
	//I_BarrieraPS308PS309_CH2		: BOOL; // 4=	
	
	I_PresenzaSupporto	: ARRAY[1..8] OF BOOL;
	I_PresenzaTelaio	: ARRAY[1..8] OF BOOL;
	I_PresenzaCentrale	: ARRAY[1..8] OF BOOL;
	I_PresenzaBundle	: ARRAY[1..8] OF BOOL; 
	
	//******************** SCHEDA IN AP200.5		
	I_AP200_5 			AT %I*: ARRAY[1..16] OF BOOL;
	//I_PresenzaSupporto[1] : BOOL;	// 1 = 
	//I_PresenzaTelaio[1]	: BOOL;	// 2 = 
	//I_PresenzaCentrale[1]	: BOOL;	// 3 = 
	//I_PresenzaBundle[1] 	: BOOL; // 4 = 
	//
	//I_PresenzaSupporto[2] : BOOL;	// 5 = 
	//I_PresenzaTelaio[2]	: BOOL;	// 6 = 
	//I_PresenzaCentrale[2]	: BOOL;	// 7 = 
	//I_PresenzaBundle[2] 	: BOOL; // 8 = 
	//
	//I_PresenzaSupporto[3] : BOOL;	// 9 = 
	//I_PresenzaTelaio[3]	: BOOL;	// 10 = 
	//I_PresenzaCentrale[3]	: BOOL;	// 11 = 
	//I_PresenzaBundle[3] 	: BOOL; // 12 = 
	//
	//I_PresenzaSupporto[4] : BOOL;	// 13 = 
	//I_PresenzaTelaio[4]	: BOOL;	// 14 = 
	//I_PresenzaCentrale[4]	: BOOL;	// 15 = 
	//I_PresenzaBundle[4] 	: BOOL; // 16 = 

	//******************** SCHEDA IN SAFETY AP200.6		
	I_AP200_6	AT %I*: ARRAY[1..4] OF BOOL;
	I_RichiestaIngressoConsolle 		AT %I* : BOOL; // 2 = Richiesta ingresso Pal CONSOLLE
	I_ResetRichiestaIngressoConsolle 	AT %I* : BOOL; // 4 = Richiesta ingresso Pal CONSOLLE
	I_PulsanteMarciaConsolle			AT %I* : BOOL; // 6 = Pulsante Marcia Pallettizzatore CH1
	I_RichiestaIngressoPS309 			AT %I* : BOOL; // 8 = Richiesta ingresso Pal PS309

	//******************** SCHEDA IN SAFETY AP200.7		
	I_AP200_7	AT %I*: ARRAY[1..4] OF BOOL;
	I_RichiestaIngressoPS306 			AT %I* : BOOL; // 2 = Richiesta ingresso Pal PS306
	I_ResetRichiestaIngressoPS306 		AT %I* : BOOL; // 4 = Reset Richiesta ingresso Pal PS306
	I_RichiestaIngressoPS307 			AT %I* : BOOL; // 6 = Richiesta ingresso Pal PS307	
	I_ResetRichiestaIngressoPS307 		AT %I* : BOOL; // 8 = Reset Richiesta ingresso Pal PS307
	
